LIN {X 0,Y 235.835,Z 423.805,A -85,B 0,C 180,E1 -19803.417,E2 -19803.417} C_VEL
LIN {X 0,Y 235.703,Z 423.051,A -85,B 0,C 180,E1 -19806.85,E2 -19806.85} C_VEL
LIN {X 0,Y 235.515,Z 422.554,A -85,B 0,C 180,E1 -19810.314,E2 -19810.314} C_VEL
LIN {X 0,Y 235.298,Z 422.298,A -85,B 0,C 180,E1 -19815.594,E2 -19815.594} C_VEL
LIN {X 0,Y 235.25,Z 422.493,A -85,B 0,C 180,E1 -19819.185,E2 -19819.185} C_VEL
LIN {X 0,Y 235.278,Z 422.982,A -85,B 0,C 180,E1 -19822.85,E2 -19822.85} C_VEL
LIN {X 0,Y 235.447,Z 423.795,A -85,B 0,C 180,E1 -19826.599,E2 -19826.599} C_VEL
LIN {X 0,Y 235.628,Z 425.005,A -85,B 0,C 180,E1 -19830.468,E2 -19830.468} C_VEL
LIN {X 0,Y 235.886,Z 426.642,A -85,B 0,C 180,E1 -19834.478,E2 -19834.478} C_VEL
LIN {X 0,Y 236.287,Z 428.755,A -85,B 0,C 180,E1 -19838.654,E2 -19838.654} C_VEL
LIN {X 0,Y 236.714,Z 431.464,A -85,B 0,C 180,E1 -19843.068,E2 -19843.068} C_VEL
LIN {X 0,Y 237.092,Z 434.077,A -85,B 0,C 180,E1 -19846.755,E2 -19846.755} C_VEL
LIN {X 0,Y 236.452,Z 434.99,A -85,B 0,C 180,E1 -19847.745,E2 -19847.745} C_VEL
LIN {X 0,Y 233.535,Z 436.791,A -85,B 0,C 180,E1 -19849.288,E2 -19849.288} C_VEL
LIN {X 0,Y 231.568,Z 438.74,A -85,B 0,C 180,E1 -19850.423,E2 -19850.423} C_VEL
LIN {X 0,Y 231.219,Z 440.688,A -85,B 0,C 180,E1 -19851.144,E2 -19851.144} C_VEL
LIN {X 0,Y 231.538,Z 441.777,A -85,B 0,C 180,E1 -19851.419,E2 -19851.419} C_VEL
LIN {X 0,Y 233.164,Z 444.382,A -85,B 0,C 180,E1 -19852.096,E2 -19852.096} C_VEL
LIN {X 0,Y 234.865,Z 448.477,A -85,B 0,C 180,E1 -19852.928,E2 -19852.928} C_VEL
LIN {X 0,Y 238.368,Z 459.348,A -85,B 0,C 180,E1 -19854.983,E2 -19854.983} C_VEL
LIN {X 0,Y 240.952,Z 471.053,A -85,B 0,C 180,E1 -19857.113,E2 -19857.113} C_VEL
LIN {X 0,Y 242.241,Z 482.421,A -85,B 0,C 180,E1 -19859.209,E2 -19859.209} C_VEL
LIN {X 0,Y 242.29,Z 492.215,A -85,B 0,C 180,E1 -19861.082,E2 -19861.082} C_VEL
LIN {X 0,Y 241.351,Z 502.224,A -85,B 0,C 180,E1 -19863.171,E2 -19863.171} C_VEL
LIN {X 0,Y 238.276,Z 511.359,A -85,B 0,C 180,E1 -19865.147,E2 -19865.147} C_VEL
LIN {X 0,Y 234.943,Z 520.47,A -85,B 0,C 180,E1 -19867.627,E2 -19867.627} C_VEL
LIN {X 0,Y 232.548,Z 527.17,A -85,B 0,C 180,E1 -19869.927,E2 -19869.927} C_VEL
LIN {X 0,Y 230.615,Z 532.669,A -85,B 0,C 180,E1 -19872.258,E2 -19872.258} C_VEL
LIN {X 0,Y 228.592,Z 537.603,A -85,B 0,C 180,E1 -19874.852,E2 -19874.852} C_VEL
LIN {X 0,Y 227.248,Z 541.454,A -85,B 0,C 180,E1 -19877.498,E2 -19877.498} C_VEL
LIN {X 0,Y 226.134,Z 545.093,A -85,B 0,C 180,E1 -19881.061,E2 -19881.061} C_VEL
LIN {X 0,Y 225.809,Z 546.282,A -85,B 0,C 180,E1 -19882.849,E2 -19882.849} C_VEL
LIN {X 0,Y 225.616,Z 547.462,A -85,B 0,C 180,E1 -19886.429,E2 -19886.429} C_VEL
LIN {X 0,Y 225.724,Z 547.477,A -85,B 0,C 180,E1 -19888.216,E2 -19888.216} C_VEL
LIN {X 0,Y 225.822,Z 547.081,A -85,B 0,C 180,E1 -19890.001,E2 -19890.001} C_VEL
LIN {X 0,Y 225.761,Z 546.237,A -85,B 0,C 180,E1 -19891.785,E2 -19891.785} C_VEL
LIN {X 0,Y 225.69,Z 543.87,A -85,B 0,C 180,E1 -19894.804,E2 -19894.804} C_VEL
LIN {X 0,Y 225.997,Z 539.926,A -85,B 0,C 180,E1 -19898.045,E2 -19898.045} C_VEL
LIN {X 0,Y 226.529,Z 535.424,A -85,B 0,C 180,E1 -19900.729,E2 -19900.729} C_VEL
LIN {X 0,Y 227.558,Z 528.552,A -85,B 0,C 180,E1 -19903.849,E2 -19903.849} C_VEL
LIN {X 0,Y 228.989,Z 521.094,A -85,B 0,C 180,E1 -19906.493,E2 -19906.493} C_VEL
LIN {X 0,Y 230.359,Z 514.102,A -85,B 0,C 180,E1 -19908.511,E2 -19908.511} C_VEL
LIN {X 0,Y 232.274,Z 504.292,A -85,B 0,C 180,E1 -19910.826,E2 -19910.826} C_VEL
LIN {X 0,Y 234.102,Z 494.094,A -85,B 0,C 180,E1 -19912.739,E2 -19912.739} C_VEL
LIN {X 0,Y 233.818,Z 485.538,A -85,B 0,C 180,E1 -19914.176,E2 -19914.176} C_VEL
LIN {X 0,Y 232.831,Z 472.863,A -85,B 0,C 180,E1 -19915.956,E2 -19915.956} C_VEL
LIN {X 0,Y 231.334,Z 461.288,A -85,B 0,C 180,E1 -19917.299,E2 -19917.299} C_VEL
LIN {X 0,Y 229.017,Z 447.664,A -85,B 0,C 180,E1 -19918.561,E2 -19918.561} C_VEL
LIN {X 0,Y 227.915,Z 441.655,A -85,B 0,C 180,E1 -19919.046,E2 -19919.046} C_VEL
LIN {X 0,Y 229.11,Z 436.101,A -85,B 0,C 180,E1 -19924.082,E2 -19924.082} C_VEL
LIN {X 0,Y 229.433,Z 434.463,A -85,B 0,C 180,E1 -19925.592,E2 -19925.592} C_VEL
LIN {X 0,Y 229.5,Z 431.075,A -85,B 0,C 180,E1 -19928.855,E2 -19928.855} C_VEL
LIN {X 0,Y 228.877,Z 427.486,A -85,B 0,C 180,E1 -19932.527,E2 -19932.527} C_VEL
LIN {X 0,Y 228.1,Z 423.047,A -85,B 0,C 180,E1 -19937.324,E2 -19937.324} C_VEL
LIN {X 0,Y 227.902,Z 422.101,A -85,B 0,C 180,E1 -19938.661,E2 -19938.661} C_VEL
LIN {X 0,Y 227.892,Z 422.093,A -85,B 0,C 180,E1 -19943.304,E2 -19943.304} C_VEL
LIN {X 0,Y 227.881,Z 422.097,A -85,B 0,C 180,E1 -19946.377,E2 -19946.377} C_VEL
LIN {X 0,Y 227.921,Z 422.092,A -85,B 0,C 180,E1 -19950.438,E2 -19950.438} C_VEL
LIN {X 0,Y 227.931,Z 422.086,A -85,B 0,C 180,E1 -19954.426,E2 -19954.426} C_VEL
LIN {X 0,Y 227.964,Z 422.087,A -85,B 0,C 180,E1 -19958.287,E2 -19958.287} C_VEL
LIN {X 0,Y 228.037,Z 422.078,A -85,B 0,C 180,E1 -19962.826,E2 -19962.826} C_VEL
LIN {X 0,Y 228.096,Z 422.068,A -85,B 0,C 180,E1 -19967.544,E2 -19967.544} C_VEL
LIN {X 0,Y 228.309,Z 422.046,A -85,B 0,C 180,E1 -19971.146,E2 -19971.146} C_VEL
LIN {X 0,Y 228.357,Z 422.041,A -85,B 0,C 180,E1 -19972.928,E2 -19972.928} C_VEL
LIN {X 0,Y 228.556,Z 422.01,A -85,B 0,C 180,E1 -19978.238,E2 -19978.238} C_VEL
LIN {X 0,Y 228.556,Z 422.011,A -85,B 0,C 180,E1 -19981.762,E2 -19981.762} C_VEL
LIN {X 0,Y 228.357,Z 422.039,A -85,B 0,C 180,E1 -19987.071,E2 -19987.071} C_VEL
LIN {X 0,Y 228.165,Z 422.063,A -85,B 0,C 180,E1 -19990.65,E2 -19990.65} C_VEL
LIN {X 0,Y 228.066,Z 422.068,A -85,B 0,C 180,E1 -19994.272,E2 -19994.272} C_VEL
LIN {X 0,Y 228.005,Z 422.061,A -85,B 0,C 180,E1 -19997.953,E2 -19997.953} C_VEL
LIN {X 0,Y 227.932,Z 422.085,A -85,B 0,C 180,E1 -20002.329,E2 -20002.329} C_VEL
LIN {X 0,Y 227.945,Z 422.092,A -85,B 0,C 180,E1 -20006.603,E2 -20006.603} C_VEL
LIN {X 0,Y 227.91,Z 422.093,A -85,B 0,C 180,E1 -20010.296,E2 -20010.296} C_VEL
LIN {X 0,Y 227.878,Z 422.087,A -85,B 0,C 180,E1 -20013.72,E2 -20013.72} C_VEL
LIN {X 0,Y 227.845,Z 422.092,A -85,B 0,C 180,E1 -20018.091,E2 -20018.091} C_VEL
LIN {X 0,Y 227.807,Z 422.109,A -85,B 0,C 180,E1 -20022.743,E2 -20022.743} C_VEL
LIN {X 0,Y 227.809,Z 422.103,A -85,B 0,C 180,E1 -20027.257,E2 -20027.257} C_VEL
LIN {X 0,Y 227.872,Z 422.088,A -85,B 0,C 180,E1 -20031.914,E2 -20031.914} C_VEL
LIN {X 0,Y 227.892,Z 422.098,A -85,B 0,C 180,E1 -20036.373,E2 -20036.373} C_VEL
LIN {X 0,Y 227.92,Z 422.092,A -85,B 0,C 180,E1 -20040.437,E2 -20040.437} C_VEL
LIN {X 0,Y 227.931,Z 422.088,A -85,B 0,C 180,E1 -20044.426,E2 -20044.426} C_VEL
LIN {X 0,Y 227.965,Z 422.09,A -85,B 0,C 180,E1 -20048.287,E2 -20048.287} C_VEL
LIN {X 0,Y 228.037,Z 422.079,A -85,B 0,C 180,E1 -20052.825,E2 -20052.825} C_VEL
LIN {X 0,Y 228.096,Z 422.071,A -85,B 0,C 180,E1 -20057.544,E2 -20057.544} C_VEL
LIN {X 0,Y 228.327,Z 422.042,A -85,B 0,C 180,E1 -20061.146,E2 -20061.146} C_VEL
LIN {X 0,Y 228.36,Z 422.037,A -85,B 0,C 180,E1 -20062.928,E2 -20062.928} C_VEL
LIN {X 0,Y 228.556,Z 422.014,A -85,B 0,C 180,E1 -20068.237,E2 -20068.237} C_VEL
LIN {X 0,Y 228.552,Z 422.016,A -85,B 0,C 180,E1 -20071.761,E2 -20071.761} C_VEL
LIN {X 0,Y 228.04,Z 422.078,A -85,B 0,C 180,E1 -20077.081,E2 -20077.081} C_VEL
LIN {X 0,Y 227.754,Z 422.115,A -85,B 0,C 180,E1 -20079.086,E2 -20079.086} C_VEL
LIN {X 0,Y 227.174,Z 425.868,A -85,B 0,C 180,E1 -20083.986,E2 -20083.986} C_VEL
LIN {X 0,Y 231.055,Z 440.646,A -85,B 0,C 180,E1 -20085.434,E2 -20085.434} C_VEL
LIN {X 0,Y 233.596,Z 452.509,A -85,B 0,C 180,E1 -20086.832,E2 -20086.832} C_VEL
LIN {X 0,Y 235.617,Z 464.141,A -85,B 0,C 180,E1 -20088.476,E2 -20088.476} C_VEL
LIN {X 0,Y 236.138,Z 469.588,A -85,B 0,C 180,E1 -20089.335,E2 -20089.335} C_VEL
LIN {X 0,Y 234.409,Z 480.31,A -85,B 0,C 180,E1 -20091.086,E2 -20091.086} C_VEL
LIN {X 0,Y 232.52,Z 490.435,A -85,B 0,C 180,E1 -20093.136,E2 -20093.136} C_VEL
LIN {X 0,Y 230.855,Z 498.791,A -85,B 0,C 180,E1 -20095.226,E2 -20095.226} C_VEL
LIN {X 0,Y 229.203,Z 507.289,A -85,B 0,C 180,E1 -20097.877,E2 -20097.877} C_VEL
LIN {X 0,Y 227.949,Z 513.581,A -85,B 0,C 180,E1 -20100.313,E2 -20100.313} C_VEL
LIN {X 0,Y 226.853,Z 519.558,A -85,B 0,C 180,E1 -20103.231,E2 -20103.231} C_VEL
LIN {X 0,Y 226.113,Z 524.157,A -85,B 0,C 180,E1 -20106.195,E2 -20106.195} C_VEL
LIN {X 0,Y 225.615,Z 527.162,A -85,B 0,C 180,E1 -20108.853,E2 -20108.853} C_VEL
LIN {X 0,Y 225.396,Z 529.228,A -85,B 0,C 180,E1 -20111.553,E2 -20111.553} C_VEL
LIN {X 0,Y 225.352,Z 530.335,A -85,B 0,C 180,E1 -20114.168,E2 -20114.168} C_VEL
LIN {X 0,Y 225.607,Z 530.602,A -85,B 0,C 180,E1 -20116.738,E2 -20116.738} C_VEL
LIN {X 0,Y 226.118,Z 530.085,A -85,B 0,C 180,E1 -20119.254,E2 -20119.254} C_VEL
LIN {X 0,Y 226.867,Z 528.825,A -85,B 0,C 180,E1 -20121.715,E2 -20121.715} C_VEL
LIN {X 0,Y 228.412,Z 525.703,A -85,B 0,C 180,E1 -20125.142,E2 -20125.142} C_VEL
LIN {X 0,Y 230.547,Z 520.882,A -85,B 0,C 180,E1 -20128.598,E2 -20128.598} C_VEL
LIN {X 0,Y 232.641,Z 515.942,A -85,B 0,C 180,E1 -20131.171,E2 -20131.171} C_VEL
LIN {X 0,Y 235.692,Z 508.399,A -85,B 0,C 180,E1 -20134.162,E2 -20134.162} C_VEL
LIN {X 0,Y 238.66,Z 500.676,A -85,B 0,C 180,E1 -20136.547,E2 -20136.547} C_VEL
LIN {X 0,Y 241.823,Z 491.575,A -85,B 0,C 180,E1 -20138.781,E2 -20138.781} C_VEL
LIN {X 0,Y 245.108,Z 480.949,A -85,B 0,C 180,E1 -20140.834,E2 -20140.834} C_VEL
LIN {X 0,Y 245.022,Z 475.384,A -85,B 0,C 180,E1 -20142.041,E2 -20142.041} C_VEL
LIN {X 0,Y 243.7,Z 465.791,A -85,B 0,C 180,E1 -20144.1,E2 -20144.1} C_VEL
LIN {X 0,Y 241.397,Z 456.441,A -85,B 0,C 180,E1 -20146.102,E2 -20146.102} C_VEL
LIN {X 0,Y 237.744,Z 445.879,A -85,B 0,C 180,E1 -20148.397,E2 -20148.397} C_VEL
LIN {X 0,Y 233.783,Z 437.563,A -85,B 0,C 180,E1 -20150.374,E2 -20150.374} C_VEL
LIN {X 0,Y 231.854,Z 433.864,A -85,B 0,C 180,E1 -20151.283,E2 -20151.283} C_VEL
LIN {X 0,Y 229.891,Z 430.981,A -85,B 0,C 180,E1 -20152.148,E2 -20152.148} C_VEL
LIN {X 0,Y 229.311,Z 429.114,A -85,B 0,C 180,E1 -20152.516,E2 -20152.516} C_VEL
LIN {X 0,Y 229.299,Z 426.856,A -85,B 0,C 180,E1 -20158.244,E2 -20158.244} C_VEL
LIN {X 0,Y 229.347,Z 426.269,A -85,B 0,C 180,E1 -20160,E2 -20160} C_VEL
LIN {X 0,Y 228.907,Z 425.375,A -85,B 0,C 180,E1 -20163.521,E2 -20163.521} C_VEL
LIN {X 0,Y 228.783,Z 424.648,A -85,B 0,C 180,E1 -20167.058,E2 -20167.058} C_VEL
LIN {X 0,Y 228.578,Z 424.194,A -85,B 0,C 180,E1 -20170.631,E2 -20170.631} C_VEL
LIN {X 0,Y 228.408,Z 424.01,A -85,B 0,C 180,E1 -20176.077,E2 -20176.077} C_VEL
LIN {X 0,Y 228.344,Z 424.262,A -85,B 0,C 180,E1 -20179.789,E2 -20179.789} C_VEL
LIN {X 0,Y 228.417,Z 424.818,A -85,B 0,C 180,E1 -20183.578,E2 -20183.578} C_VEL
LIN {X 0,Y 228.565,Z 425.728,A -85,B 0,C 180,E1 -20187.466,E2 -20187.466} C_VEL
LIN {X 0,Y 228.774,Z 427.042,A -85,B 0,C 180,E1 -20191.483,E2 -20191.483} C_VEL
LIN {X 0,Y 229.06,Z 428.821,A -85,B 0,C 180,E1 -20195.659,E2 -20195.659} C_VEL
LIN {X 0,Y 229.485,Z 431.109,A -85,B 0,C 180,E1 -20200.039,E2 -20200.039} C_VEL
LIN {X 0,Y 229.946,Z 434.016,A -85,B 0,C 180,E1 -20204.666,E2 -20204.666} C_VEL
LIN {X 0,Y 230.259,Z 436.263,A -85,B 0,C 180,E1 -20207.819,E2 -20207.819} C_VEL
LIN {X 0,Y 230.501,Z 438.815,A -85,B 0,C 180,E1 -20210.885,E2 -20210.885} C_VEL
LIN {X 0,Y 231.538,Z 441.777,A -85,B 0,C 180,E1 -20211.419,E2 -20211.419} C_VEL
LIN {X 0,Y 233.041,Z 446.441,A -85,B 0,C 180,E1 -20212.239,E2 -20212.239} C_VEL
LIN {X 0,Y 233.732,Z 451.625,A -85,B 0,C 180,E1 -20212.942,E2 -20212.942} C_VEL
LIN {X 0,Y 233.917,Z 462.354,A -85,B 0,C 180,E1 -20214.29,E2 -20214.29} C_VEL
LIN {X 0,Y 234.213,Z 467.417,A -85,B 0,C 180,E1 -20215.082,E2 -20215.082} C_VEL
LIN {X 0,Y 234.461,Z 468.99,A -85,B 0,C 180,E1 -20215.38,E2 -20215.38} C_VEL
LIN {X 0,Y 235.858,Z 478.402,A -85,B 0,C 180,E1 -20217.22,E2 -20217.22} C_VEL
LIN {X 0,Y 236.337,Z 487.526,A -85,B 0,C 180,E1 -20219.049,E2 -20219.049} C_VEL
LIN {X 0,Y 235.81,Z 497.788,A -85,B 0,C 180,E1 -20221.194,E2 -20221.194} C_VEL
LIN {X 0,Y 235.062,Z 503.127,A -85,B 0,C 180,E1 -20222.393,E2 -20222.393} C_VEL
LIN {X 0,Y 231.906,Z 512.029,A -85,B 0,C 180,E1 -20224.416,E2 -20224.416} C_VEL
LIN {X 0,Y 228.479,Z 520.817,A -85,B 0,C 180,E1 -20226.91,E2 -20226.91} C_VEL
LIN {X 0,Y 225.831,Z 527.661,A -85,B 0,C 180,E1 -20229.377,E2 -20229.377} C_VEL
LIN {X 0,Y 223.854,Z 532.868,A -85,B 0,C 180,E1 -20231.703,E2 -20231.703} C_VEL
LIN {X 0,Y 221.737,Z 537.702,A -85,B 0,C 180,E1 -20234.372,E2 -20234.372} C_VEL
LIN {X 0,Y 220.275,Z 541.458,A -85,B 0,C 180,E1 -20237.096,E2 -20237.096} C_VEL
LIN {X 0,Y 219.602,Z 543.43,A -85,B 0,C 180,E1 -20238.93,E2 -20238.93} C_VEL
LIN {X 0,Y 219.087,Z 544.981,A -85,B 0,C 180,E1 -20240.771,E2 -20240.771} C_VEL
LIN {X 0,Y 218.568,Z 546.843,A -85,B 0,C 180,E1 -20244.465,E2 -20244.465} C_VEL
LIN {X 0,Y 218.635,Z 547.175,A -85,B 0,C 180,E1 -20248.159,E2 -20248.159} C_VEL
LIN {X 0,Y 218.754,Z 546.708,A -85,B 0,C 180,E1 -20250.001,E2 -20250.001} C_VEL
LIN {X 0,Y 218.671,Z 545.825,A -85,B 0,C 180,E1 -20251.842,E2 -20251.842} C_VEL
LIN {X 0,Y 218.593,Z 543.659,A -85,B 0,C 180,E1 -20254.664,E2 -20254.664} C_VEL
LIN {X 0,Y 218.813,Z 540.59,A -85,B 0,C 180,E1 -20257.382,E2 -20257.382} C_VEL
LIN {X 0,Y 219.292,Z 536.374,A -85,B 0,C 180,E1 -20260.153,E2 -20260.153} C_VEL
LIN {X 0,Y 220.229,Z 529.927,A -85,B 0,C 180,E1 -20263.378,E2 -20263.378} C_VEL
LIN {X 0,Y 221.655,Z 522.877,A -85,B 0,C 180,E1 -20266.108,E2 -20266.108} C_VEL
LIN {X 0,Y 223.291,Z 514.581,A -85,B 0,C 180,E1 -20268.665,E2 -20268.665} C_VEL
LIN {X 0,Y 225.195,Z 505.019,A -85,B 0,C 180,E1 -20271.033,E2 -20271.033} C_VEL
LIN {X 0,Y 227.088,Z 495.116,A -85,B 0,C 180,E1 -20273,E2 -20273} C_VEL
LIN {X 0,Y 227.041,Z 488.306,A -85,B 0,C 180,E1 -20274.207,E2 -20274.207} C_VEL
LIN {X 0,Y 226.276,Z 476.943,A -85,B 0,C 180,E1 -20275.972,E2 -20275.972} C_VEL
LIN {X 0,Y 224.921,Z 464.647,A -85,B 0,C 180,E1 -20277.548,E2 -20277.548} C_VEL
LIN {X 0,Y 222.726,Z 450.893,A -85,B 0,C 180,E1 -20278.964,E2 -20278.964} C_VEL
LIN {X 0,Y 221.002,Z 441.394,A -85,B 0,C 180,E1 -20279.779,E2 -20279.779} C_VEL
LIN {X 0,Y 222.16,Z 436.145,A -85,B 0,C 180,E1 -20284.711,E2 -20284.711} C_VEL
LIN {X 0,Y 222.469,Z 432.936,A -85,B 0,C 180,E1 -20287.835,E2 -20287.835} C_VEL
LIN {X 0,Y 222.174,Z 430.256,A -85,B 0,C 180,E1 -20290.607,E2 -20290.607} C_VEL
LIN {X 0,Y 221.536,Z 426.856,A -85,B 0,C 180,E1 -20294.261,E2 -20294.261} C_VEL
LIN {X 0,Y 220.878,Z 422.977,A -85,B 0,C 180,E1 -20298.787,E2 -20298.787} C_VEL
LIN {X 0,Y 220.826,Z 422.977,A -85,B 0,C 180,E1 -20302.793,E2 -20302.793} C_VEL
LIN {X 0,Y 220.82,Z 422.982,A -85,B 0,C 180,E1 -20307.244,E2 -20307.244} C_VEL
LIN {X 0,Y 220.839,Z 422.97,A -85,B 0,C 180,E1 -20311.487,E2 -20311.487} C_VEL
LIN {X 0,Y 220.87,Z 422.971,A -85,B 0,C 180,E1 -20315.565,E2 -20315.565} C_VEL
LIN {X 0,Y 220.895,Z 422.968,A -85,B 0,C 180,E1 -20319.514,E2 -20319.514} C_VEL
LIN {X 0,Y 221.019,Z 422.954,A -85,B 0,C 180,E1 -20323.37,E2 -20323.37} C_VEL
LIN {X 0,Y 221.114,Z 422.939,A -85,B 0,C 180,E1 -20329.006,E2 -20329.006} C_VEL
LIN {X 0,Y 221.292,Z 422.919,A -85,B 0,C 180,E1 -20332.702,E2 -20332.702} C_VEL
LIN {X 0,Y 221.514,Z 422.887,A -85,B 0,C 180,E1 -20338.182,E2 -20338.182} C_VEL
LIN {X 0,Y 221.514,Z 422.888,A -85,B 0,C 180,E1 -20341.818,E2 -20341.818} C_VEL
LIN {X 0,Y 221.292,Z 422.918,A -85,B 0,C 180,E1 -20347.298,E2 -20347.298} C_VEL
LIN {X 0,Y 221.114,Z 422.94,A -85,B 0,C 180,E1 -20350.994,E2 -20350.994} C_VEL
LIN {X 0,Y 221.018,Z 422.936,A -85,B 0,C 180,E1 -20356.63,E2 -20356.63} C_VEL
LIN {X 0,Y 220.894,Z 422.955,A -85,B 0,C 180,E1 -20360.486,E2 -20360.486} C_VEL
LIN {X 0,Y 220.869,Z 422.969,A -85,B 0,C 180,E1 -20364.435,E2 -20364.435} C_VEL
LIN {X 0,Y 220.839,Z 422.977,A -85,B 0,C 180,E1 -20368.513,E2 -20368.513} C_VEL
LIN {X 0,Y 220.819,Z 422.969,A -85,B 0,C 180,E1 -20372.756,E2 -20372.756} C_VEL
LIN {X 0,Y 220.811,Z 422.967,A -85,B 0,C 180,E1 -20377.278,E2 -20377.278} C_VEL
LIN {X 0,Y 220.796,Z 422.975,A -85,B 0,C 180,E1 -20380.188,E2 -20380.188} C_VEL
LIN {X 0,Y 220.769,Z 422.986,A -85,B 0,C 180,E1 -20384.455,E2 -20384.455} C_VEL
LIN {X 0,Y 220.773,Z 422.979,A -85,B 0,C 180,E1 -20388.048,E2 -20388.048} C_VEL
LIN {X 0,Y 220.834,Z 422.969,A -85,B 0,C 180,E1 -20392.794,E2 -20392.794} C_VEL
LIN {X 0,Y 220.826,Z 422.976,A -85,B 0,C 180,E1 -20397.245,E2 -20397.245} C_VEL
LIN {X 0,Y 220.838,Z 422.969,A -85,B 0,C 180,E1 -20401.486,E2 -20401.486} C_VEL
LIN {X 0,Y 220.87,Z 422.969,A -85,B 0,C 180,E1 -20405.565,E2 -20405.565} C_VEL
LIN {X 0,Y 220.895,Z 422.967,A -85,B 0,C 180,E1 -20409.514,E2 -20409.514} C_VEL
LIN {X 0,Y 221.019,Z 422.951,A -85,B 0,C 180,E1 -20413.37,E2 -20413.37} C_VEL
LIN {X 0,Y 221.119,Z 422.938,A -85,B 0,C 180,E1 -20419.006,E2 -20419.006} C_VEL
LIN {X 0,Y 221.313,Z 422.916,A -85,B 0,C 180,E1 -20422.702,E2 -20422.702} C_VEL
LIN {X 0,Y 221.514,Z 422.89,A -85,B 0,C 180,E1 -20428.181,E2 -20428.181} C_VEL
LIN {X 0,Y 221.508,Z 422.894,A -85,B 0,C 180,E1 -20431.817,E2 -20431.817} C_VEL
LIN {X 0,Y 220.963,Z 422.96,A -85,B 0,C 180,E1 -20437.309,E2 -20437.309} C_VEL
LIN {X 0,Y 220.683,Z 423.074,A -85,B 0,C 180,E1 -20439.162,E2 -20439.162} C_VEL
LIN {X 0,Y 220.175,Z 426.153,A -85,B 0,C 180,E1 -20443.262,E2 -20443.262} C_VEL
LIN {X 0,Y 223.641,Z 439.187,A -85,B 0,C 180,E1 -20444.56,E2 -20444.56} C_VEL
LIN {X 0,Y 226.316,Z 451.122,A -85,B 0,C 180,E1 -20445.997,E2 -20445.997} C_VEL
LIN {X 0,Y 228.418,Z 462.946,A -85,B 0,C 180,E1 -20447.687,E2 -20447.687} C_VEL
LIN {X 0,Y 229.33,Z 469.548,A -85,B 0,C 180,E1 -20448.77,E2 -20448.77} C_VEL
LIN {X 0,Y 227.654,Z 480.216,A -85,B 0,C 180,E1 -20450.557,E2 -20450.557} C_VEL
LIN {X 0,Y 225.684,Z 490.407,A -85,B 0,C 180,E1 -20452.666,E2 -20452.666} C_VEL
LIN {X 0,Y 223.941,Z 498.898,A -85,B 0,C 180,E1 -20454.838,E2 -20454.838} C_VEL
LIN {X 0,Y 222.181,Z 507.691,A -85,B 0,C 180,E1 -20457.663,E2 -20457.663} C_VEL
LIN {X 0,Y 220.66,Z 515.118,A -85,B 0,C 180,E1 -20460.689,E2 -20460.689} C_VEL
LIN {X 0,Y 219.62,Z 520.768,A -85,B 0,C 180,E1 -20463.693,E2 -20463.693} C_VEL
LIN {X 0,Y 218.913,Z 524.943,A -85,B 0,C 180,E1 -20466.621,E2 -20466.621} C_VEL
LIN {X 0,Y 218.374,Z 528.377,A -85,B 0,C 180,E1 -20470.064,E2 -20470.064} C_VEL
LIN {X 0,Y 218.251,Z 529.922,A -85,B 0,C 180,E1 -20472.548,E2 -20472.548} C_VEL
LIN {X 0,Y 218.314,Z 530.772,A -85,B 0,C 180,E1 -20475.089,E2 -20475.089} C_VEL
LIN {X 0,Y 218.659,Z 530.86,A -85,B 0,C 180,E1 -20477.666,E2 -20477.666} C_VEL
LIN {X 0,Y 219.313,Z 530.146,A -85,B 0,C 180,E1 -20480.271,E2 -20480.271} C_VEL
LIN {X 0,Y 220.258,Z 528.623,A -85,B 0,C 180,E1 -20482.909,E2 -20482.909} C_VEL
LIN {X 0,Y 221.527,Z 526.216,A -85,B 0,C 180,E1 -20485.572,E2 -20485.572} C_VEL
LIN {X 0,Y 223.753,Z 521.546,A -85,B 0,C 180,E1 -20489.085,E2 -20489.085} C_VEL
LIN {X 0,Y 226.456,Z 515.596,A -85,B 0,C 180,E1 -20492.256,E2 -20492.256} C_VEL
LIN {X 0,Y 229.341,Z 508.93,A -85,B 0,C 180,E1 -20494.958,E2 -20494.958} C_VEL
LIN {X 0,Y 232.287,Z 501.744,A -85,B 0,C 180,E1 -20497.259,E2 -20497.259} C_VEL
LIN {X 0,Y 235.51,Z 493.129,A -85,B 0,C 180,E1 -20499.474,E2 -20499.474} C_VEL
LIN {X 0,Y 238.667,Z 483.566,A -85,B 0,C 180,E1 -20501.434,E2 -20501.434} C_VEL
LIN {X 0,Y 239.088,Z 481.667,A -85,B 0,C 180,E1 -20501.801,E2 -20501.801} C_VEL
LIN {X 0,Y 238.557,Z 473.342,A -85,B 0,C 180,E1 -20503.747,E2 -20503.747} C_VEL
LIN {X 0,Y 237.059,Z 464.122,A -85,B 0,C 180,E1 -20505.843,E2 -20505.843} C_VEL
LIN {X 0,Y 234.087,Z 453.725,A -85,B 0,C 180,E1 -20508.268,E2 -20508.268} C_VEL
LIN {X 0,Y 231.492,Z 446.805,A -85,B 0,C 180,E1 -20509.947,E2 -20509.947} C_VEL
LIN {X 0,Y 227.917,Z 439.271,A -85,B 0,C 180,E1 -20511.929,E2 -20511.929} C_VEL
LIN {X 0,Y 225.984,Z 436.076,A -85,B 0,C 180,E1 -20512.91,E2 -20512.91} C_VEL
LIN {X 0,Y 225.03,Z 434.44,A -85,B 0,C 180,E1 -20513.387,E2 -20513.387} C_VEL
LIN {X 0,Y 222.916,Z 431.575,A -85,B 0,C 180,E1 -20514.403,E2 -20514.403} C_VEL
LIN {X 0,Y 222.29,Z 429.592,A -85,B 0,C 180,E1 -20514.899,E2 -20514.899} C_VEL
LIN {X 0,Y 222.364,Z 428.394,A -85,B 0,C 180,E1 -20518.189,E2 -20518.189} C_VEL
LIN {X 0,Y 222.415,Z 427.824,A -85,B 0,C 180,E1 -20520,E2 -20520} C_VEL
LIN {X 0,Y 221.969,Z 426.951,A -85,B 0,C 180,E1 -20523.631,E2 -20523.631} C_VEL
LIN {X 0,Y 221.856,Z 426.256,A -85,B 0,C 180,E1 -20527.28,E2 -20527.28} C_VEL
LIN {X 0,Y 221.645,Z 425.849,A -85,B 0,C 180,E1 -20530.968,E2 -20530.968} C_VEL
LIN {X 0,Y 221.503,Z 425.734,A -85,B 0,C 180,E1 -20536.592,E2 -20536.592} C_VEL
LIN {X 0,Y 221.45,Z 426.047,A -85,B 0,C 180,E1 -20540.432,E2 -20540.432} C_VEL
LIN {X 0,Y 221.528,Z 426.682,A -85,B 0,C 180,E1 -20544.358,E2 -20544.358} C_VEL
LIN {X 0,Y 221.695,Z 427.69,A -85,B 0,C 180,E1 -20548.393,E2 -20548.393} C_VEL
LIN {X 0,Y 221.917,Z 429.133,A -85,B 0,C 180,E1 -20552.574,E2 -20552.574} C_VEL
LIN {X 0,Y 222.358,Z 431.469,A -85,B 0,C 180,E1 -20557.8,E2 -20557.8} C_VEL
LIN {X 0,Y 222.669,Z 433.515,A -85,B 0,C 180,E1 -20561.515,E2 -20561.515} C_VEL
LIN {X 0,Y 223.123,Z 436.466,A -85,B 0,C 180,E1 -20566.136,E2 -20566.136} C_VEL
LIN {X 0,Y 223.334,Z 438.161,A -85,B 0,C 180,E1 -20568.52,E2 -20568.52} C_VEL
LIN {X 0,Y 224.515,Z 441.421,A -85,B 0,C 180,E1 -20569.213,E2 -20569.213} C_VEL
LIN {X 0,Y 226.615,Z 444.574,A -85,B 0,C 180,E1 -20570.187,E2 -20570.187} C_VEL
LIN {X 0,Y 228.466,Z 448.596,A -85,B 0,C 180,E1 -20571.171,E2 -20571.171} C_VEL
LIN {X 0,Y 230.722,Z 454.495,A -85,B 0,C 180,E1 -20572.468,E2 -20572.468} C_VEL
LIN {X 0,Y 233.238,Z 463.05,A -85,B 0,C 180,E1 -20574.214,E2 -20574.214} C_VEL
LIN {X 0,Y 234.461,Z 468.99,A -85,B 0,C 180,E1 -20575.38,E2 -20575.38} C_VEL
LIN {X 0,Y 234.759,Z 473.886,A -85,B 0,C 180,E1 -20576.215,E2 -20576.215} C_VEL
LIN {X 0,Y 233.953,Z 479.09,A -85,B 0,C 180,E1 -20576.937,E2 -20576.937} C_VEL
LIN {X 0,Y 231.165,Z 489.229,A -85,B 0,C 180,E1 -20578.37,E2 -20578.37} C_VEL
LIN {X 0,Y 230.115,Z 493.949,A -85,B 0,C 180,E1 -20579.229,E2 -20579.229} C_VEL
LIN {X 0,Y 229.937,Z 495.417,A -85,B 0,C 180,E1 -20579.55,E2 -20579.55} C_VEL
LIN {X 0,Y 228.798,Z 504.005,A -85,B 0,C 180,E1 -20581.569,E2 -20581.569} C_VEL
LIN {X 0,Y 225.553,Z 512.702,A -85,B 0,C 180,E1 -20583.641,E2 -20583.641} C_VEL
LIN {X 0,Y 221.978,Z 521.337,A -85,B 0,C 180,E1 -20586.193,E2 -20586.193} C_VEL
LIN {X 0,Y 219.137,Z 528.2,A -85,B 0,C 180,E1 -20588.795,E2 -20588.795} C_VEL
LIN {X 0,Y 217.12,Z 533.108,A -85,B 0,C 180,E1 -20591.115,E2 -20591.115} C_VEL
LIN {X 0,Y 214.902,Z 537.812,A -85,B 0,C 180,E1 -20593.861,E2 -20593.861} C_VEL
LIN {X 0,Y 213.315,Z 541.464,A -85,B 0,C 180,E1 -20596.667,E2 -20596.667} C_VEL
LIN {X 0,Y 212.609,Z 543.384,A -85,B 0,C 180,E1 -20598.561,E2 -20598.561} C_VEL
LIN {X 0,Y 211.669,Z 545.931,A -85,B 0,C 180,E1 -20602.369,E2 -20602.369} C_VEL
LIN {X 0,Y 211.437,Z 546.946,A -85,B 0,C 180,E1 -20606.189,E2 -20606.189} C_VEL
LIN {X 0,Y 211.547,Z 546.843,A -85,B 0,C 180,E1 -20608.097,E2 -20608.097} C_VEL
LIN {X 0,Y 211.687,Z 546.332,A -85,B 0,C 180,E1 -20610.001,E2 -20610.001} C_VEL
LIN {X 0,Y 211.584,Z 545.41,A -85,B 0,C 180,E1 -20611.904,E2 -20611.904} C_VEL
LIN {X 0,Y 211.508,Z 543.417,A -85,B 0,C 180,E1 -20614.55,E2 -20614.55} C_VEL
LIN {X 0,Y 211.743,Z 540.009,A -85,B 0,C 180,E1 -20617.63,E2 -20617.63} C_VEL
LIN {X 0,Y 212.269,Z 535.701,A -85,B 0,C 180,E1 -20620.493,E2 -20620.493} C_VEL
LIN {X 0,Y 213.078,Z 530.167,A -85,B 0,C 180,E1 -20623.35,E2 -20623.35} C_VEL
LIN {X 0,Y 214.527,Z 523.266,A -85,B 0,C 180,E1 -20626.169,E2 -20626.169} C_VEL
LIN {X 0,Y 216.293,Z 514.598,A -85,B 0,C 180,E1 -20628.962,E2 -20628.962} C_VEL
LIN {X 0,Y 218.113,Z 505.73,A -85,B 0,C 180,E1 -20631.254,E2 -20631.254} C_VEL
LIN {X 0,Y 220.25,Z 494.853,A -85,B 0,C 180,E1 -20633.508,E2 -20633.508} C_VEL
LIN {X 0,Y 219.875,Z 484.523,A -85,B 0,C 180,E1 -20635.372,E2 -20635.372} C_VEL
LIN {X 0,Y 219.032,Z 473.317,A -85,B 0,C 180,E1 -20637.07,E2 -20637.07} C_VEL
LIN {X 0,Y 217.436,Z 460.354,A -85,B 0,C 180,E1 -20638.69,E2 -20638.69} C_VEL
LIN {X 0,Y 215.113,Z 447.007,A -85,B 0,C 180,E1 -20640.016,E2 -20640.016} C_VEL
LIN {X 0,Y 214.084,Z 441.156,A -85,B 0,C 180,E1 -20640.516,E2 -20640.516} C_VEL
LIN {X 0,Y 215.194,Z 436.293,A -85,B 0,C 180,E1 -20645.267,E2 -20645.267} C_VEL
LIN {X 0,Y 215.402,Z 433.154,A -85,B 0,C 180,E1 -20648.458,E2 -20648.458} C_VEL
LIN {X 0,Y 215.022,Z 430.532,A -85,B 0,C 180,E1 -20651.257,E2 -20651.257} C_VEL
LIN {X 0,Y 214.361,Z 427.072,A -85,B 0,C 180,E1 -20655.146,E2 -20655.146} C_VEL
LIN {X 0,Y 213.799,Z 423.86,A -85,B 0,C 180,E1 -20659.118,E2 -20659.118} C_VEL
LIN {X 0,Y 213.746,Z 423.852,A -85,B 0,C 180,E1 -20663.712,E2 -20663.712} C_VEL
LIN {X 0,Y 213.797,Z 423.855,A -85,B 0,C 180,E1 -20668.725,E2 -20668.725} C_VEL
LIN {X 0,Y 213.828,Z 423.841,A -85,B 0,C 180,E1 -20672.603,E2 -20672.603} C_VEL
LIN {X 0,Y 213.854,Z 423.846,A -85,B 0,C 180,E1 -20676.953,E2 -20676.953} C_VEL
LIN {X 0,Y 213.946,Z 423.832,A -85,B 0,C 180,E1 -20682.804,E2 -20682.804} C_VEL
LIN {X 0,Y 213.983,Z 423.83,A -85,B 0,C 180,E1 -20686.708,E2 -20686.708} C_VEL
LIN {X 0,Y 214.17,Z 423.804,A -85,B 0,C 180,E1 -20690.556,E2 -20690.556} C_VEL
LIN {X 0,Y 214.23,Z 423.798,A -85,B 0,C 180,E1 -20692.46,E2 -20692.46} C_VEL
LIN {X 0,Y 214.447,Z 423.767,A -85,B 0,C 180,E1 -20698.122,E2 -20698.122} C_VEL
LIN {X 0,Y 214.548,Z 423.757,A -85,B 0,C 180,E1 -20700,E2 -20700} C_VEL
LIN {X 0,Y 214.447,Z 423.769,A -85,B 0,C 180,E1 -20701.878,E2 -20701.878} C_VEL
LIN {X 0,Y 214.23,Z 423.796,A -85,B 0,C 180,E1 -20707.54,E2 -20707.54} C_VEL
LIN {X 0,Y 214.047,Z 423.818,A -85,B 0,C 180,E1 -20711.362,E2 -20711.362} C_VEL
LIN {X 0,Y 213.935,Z 423.822,A -85,B 0,C 180,E1 -20715.237,E2 -20715.237} C_VEL
LIN {X 0,Y 213.842,Z 423.829,A -85,B 0,C 180,E1 -20719.187,E2 -20719.187} C_VEL
LIN {X 0,Y 213.849,Z 423.843,A -85,B 0,C 180,E1 -20723.227,E2 -20723.227} C_VEL
LIN {X 0,Y 213.831,Z 423.848,A -85,B 0,C 180,E1 -20727.45,E2 -20727.45} C_VEL
LIN {X 0,Y 213.779,Z 423.848,A -85,B 0,C 180,E1 -20731.736,E2 -20731.736} C_VEL
LIN {X 0,Y 213.745,Z 423.838,A -85,B 0,C 180,E1 -20736.288,E2 -20736.288} C_VEL
LIN {X 0,Y 213.712,Z 423.861,A -85,B 0,C 180,E1 -20741.125,E2 -20741.125} C_VEL
LIN {X 0,Y 213.704,Z 423.863,A -85,B 0,C 180,E1 -20743.679,E2 -20743.679} C_VEL
LIN {X 0,Y 213.704,Z 423.864,A -85,B 0,C 180,E1 -20746.345,E2 -20746.345} C_VEL
LIN {X 0,Y 213.737,Z 423.847,A -85,B 0,C 180,E1 -20751.336,E2 -20751.336} C_VEL
LIN {X 0,Y 213.771,Z 423.854,A -85,B 0,C 180,E1 -20756.02,E2 -20756.02} C_VEL
LIN {X 0,Y 213.782,Z 423.853,A -85,B 0,C 180,E1 -20760.454,E2 -20760.454} C_VEL
LIN {X 0,Y 213.804,Z 423.849,A -85,B 0,C 180,E1 -20764.701,E2 -20764.701} C_VEL
LIN {X 0,Y 213.816,Z 423.85,A -85,B 0,C 180,E1 -20768.803,E2 -20768.803} C_VEL
LIN {X 0,Y 213.946,Z 423.834,A -85,B 0,C 180,E1 -20772.803,E2 -20772.803} C_VEL
LIN {X 0,Y 213.983,Z 423.831,A -85,B 0,C 180,E1 -20776.708,E2 -20776.708} C_VEL
LIN {X 0,Y 214.199,Z 423.805,A -85,B 0,C 180,E1 -20780.557,E2 -20780.557} C_VEL
LIN {X 0,Y 214.25,Z 423.797,A -85,B 0,C 180,E1 -20782.46,E2 -20782.46} C_VEL
LIN {X 0,Y 214.447,Z 423.77,A -85,B 0,C 180,E1 -20788.121,E2 -20788.121} C_VEL
LIN {X 0,Y 214.551,Z 423.762,A -85,B 0,C 180,E1 -20789.999,E2 -20789.999} C_VEL
LIN {X 0,Y 214.44,Z 423.774,A -85,B 0,C 180,E1 -20791.877,E2 -20791.877} C_VEL
LIN {X 0,Y 213.894,Z 423.84,A -85,B 0,C 180,E1 -20797.551,E2 -20797.551} C_VEL
LIN {X 0,Y 213.627,Z 424.046,A -85,B 0,C 180,E1 -20799.265,E2 -20799.265} C_VEL
LIN {X 0,Y 213.177,Z 426.423,A -85,B 0,C 180,E1 -20802.494,E2 -20802.494} C_VEL
LIN {X 0,Y 217.086,Z 441.141,A -85,B 0,C 180,E1 -20804.052,E2 -20804.052} C_VEL
LIN {X 0,Y 219.678,Z 452.86,A -85,B 0,C 180,E1 -20805.541,E2 -20805.541} C_VEL
LIN {X 0,Y 221.665,Z 464.481,A -85,B 0,C 180,E1 -20807.291,E2 -20807.291} C_VEL
LIN {X 0,Y 222.437,Z 471.003,A -85,B 0,C 180,E1 -20808.418,E2 -20808.418} C_VEL
LIN {X 0,Y 220.623,Z 481.552,A -85,B 0,C 180,E1 -20810.268,E2 -20810.268} C_VEL
LIN {X 0,Y 218.653,Z 491.445,A -85,B 0,C 180,E1 -20812.416,E2 -20812.416} C_VEL
LIN {X 0,Y 216.692,Z 500.689,A -85,B 0,C 180,E1 -20814.937,E2 -20814.937} C_VEL
LIN {X 0,Y 215.068,Z 508.475,A -85,B 0,C 180,E1 -20817.577,E2 -20817.577} C_VEL
LIN {X 0,Y 213.697,Z 514.916,A -85,B 0,C 180,E1 -20820.293,E2 -20820.293} C_VEL
LIN {X 0,Y 212.695,Z 520.051,A -85,B 0,C 180,E1 -20823.01,E2 -20823.01} C_VEL
LIN {X 0,Y 211.795,Z 525.251,A -85,B 0,C 180,E1 -20826.675,E2 -20826.675} C_VEL
LIN {X 0,Y 211.285,Z 528.555,A -85,B 0,C 180,E1 -20830.088,E2 -20830.088} C_VEL
LIN {X 0,Y 211.14,Z 530.265,A -85,B 0,C 180,E1 -20832.921,E2 -20832.921} C_VEL
LIN {X 0,Y 211.285,Z 531.09,A -85,B 0,C 180,E1 -20835.691,E2 -20835.691} C_VEL
LIN {X 0,Y 212.031,Z 530.836,A -85,B 0,C 180,E1 -20839.671,E2 -20839.671} C_VEL
LIN {X 0,Y 212.932,Z 529.638,A -85,B 0,C 180,E1 -20842.384,E2 -20842.384} C_VEL
LIN {X 0,Y 214.743,Z 526.557,A -85,B 0,C 180,E1 -20846.195,E2 -20846.195} C_VEL
LIN {X 0,Y 217.087,Z 522.051,A -85,B 0,C 180,E1 -20849.727,E2 -20849.727} C_VEL
LIN {X 0,Y 219.843,Z 516.42,A -85,B 0,C 180,E1 -20852.885,E2 -20852.885} C_VEL
LIN {X 0,Y 223.221,Z 509.122,A -85,B 0,C 180,E1 -20855.928,E2 -20855.928} C_VEL
LIN {X 0,Y 226.638,Z 501.223,A -85,B 0,C 180,E1 -20858.478,E2 -20858.478} C_VEL
LIN {X 0,Y 230.434,Z 491.296,A -85,B 0,C 180,E1 -20860.988,E2 -20860.988} C_VEL
LIN {X 0,Y 232.865,Z 484.289,A -85,B 0,C 180,E1 -20862.434,E2 -20862.434} C_VEL
LIN {X 0,Y 232.744,Z 476.985,A -85,B 0,C 180,E1 -20864.231,E2 -20864.231} C_VEL
LIN {X 0,Y 231.604,Z 468.053,A -85,B 0,C 180,E1 -20866.398,E2 -20866.398} C_VEL
LIN {X 0,Y 229.109,Z 458.055,A -85,B 0,C 180,E1 -20868.907,E2 -20868.907} C_VEL
LIN {X 0,Y 225.674,Z 448.377,A -85,B 0,C 180,E1 -20871.445,E2 -20871.445} C_VEL
LIN {X 0,Y 221.431,Z 440.186,A -85,B 0,C 180,E1 -20873.965,E2 -20873.965} C_VEL
LIN {X 0,Y 219.249,Z 436.795,A -85,B 0,C 180,E1 -20875.211,E2 -20875.211} C_VEL
LIN {X 0,Y 218.487,Z 435.333,A -85,B 0,C 180,E1 -20875.671,E2 -20875.671} C_VEL
LIN {X 0,Y 216.276,Z 432.694,A -85,B 0,C 180,E1 -20876.857,E2 -20876.857} C_VEL
LIN {X 0,Y 215.382,Z 430.14,A -85,B 0,C 180,E1 -20877.546,E2 -20877.546} C_VEL
LIN {X 0,Y 215.508,Z 429.371,A -85,B 0,C 180,E1 -20880,E2 -20880} C_VEL
LIN {X 0,Y 215.037,Z 428.538,A -85,B 0,C 180,E1 -20883.748,E2 -20883.748} C_VEL
LIN {X 0,Y 214.926,Z 427.872,A -85,B 0,C 180,E1 -20887.516,E2 -20887.516} C_VEL
LIN {X 0,Y 214.715,Z 427.506,A -85,B 0,C 180,E1 -20891.326,E2 -20891.326} C_VEL
LIN {X 0,Y 214.583,Z 427.422,A -85,B 0,C 180,E1 -20895.19,E2 -20895.19} C_VEL
LIN {X 0,Y 214.548,Z 427.634,A -85,B 0,C 180,E1 -20899.122,E2 -20899.122} C_VEL
LIN {X 0,Y 214.637,Z 428.242,A -85,B 0,C 180,E1 -20903.537,E2 -20903.537} C_VEL
LIN {X 0,Y 214.782,Z 429.258,A -85,B 0,C 180,E1 -20907.937,E2 -20907.937} C_VEL
LIN {X 0,Y 214.969,Z 430.494,A -85,B 0,C 180,E1 -20911.788,E2 -20911.788} C_VEL
LIN {X 0,Y 215.234,Z 432.211,A -85,B 0,C 180,E1 -20915.998,E2 -20915.998} C_VEL
LIN {X 0,Y 215.686,Z 434.544,A -85,B 0,C 180,E1 -20920.669,E2 -20920.669} C_VEL
LIN {X 0,Y 216.116,Z 437.631,A -85,B 0,C 180,E1 -20925.748,E2 -20925.748} C_VEL
LIN {X 0,Y 217.425,Z 441.015,A -85,B 0,C 180,E1 -20926.629,E2 -20926.629} C_VEL
LIN {X 0,Y 219.699,Z 444.17,A -85,B 0,C 180,E1 -20927.83,E2 -20927.83} C_VEL
LIN {X 0,Y 221.426,Z 447.891,A -85,B 0,C 180,E1 -20928.861,E2 -20928.861} C_VEL
LIN {X 0,Y 222.698,Z 450.113,A -85,B 0,C 180,E1 -20929.54,E2 -20929.54} C_VEL
LIN {X 0,Y 225.744,Z 457.855,A -85,B 0,C 180,E1 -20931.491,E2 -20931.491} C_VEL
LIN {X 0,Y 228.199,Z 467.369,A -85,B 0,C 180,E1 -20933.571,E2 -20933.571} C_VEL
LIN {X 0,Y 229.877,Z 478.673,A -85,B 0,C 180,E1 -20935.957,E2 -20935.957} C_VEL
LIN {X 0,Y 230.32,Z 488.518,A -85,B 0,C 180,E1 -20938.037,E2 -20938.037} C_VEL
LIN {X 0,Y 229.937,Z 495.417,A -85,B 0,C 180,E1 -20939.55,E2 -20939.55} C_VEL
LIN {X 0,Y 229.312,Z 498.428,A -85,B 0,C 180,E1 -20940.171,E2 -20940.171} C_VEL
LIN {X 0,Y 228.066,Z 501.453,A -85,B 0,C 180,E1 -20940.727,E2 -20940.727} C_VEL
LIN {X 0,Y 224.459,Z 507.306,A -85,B 0,C 180,E1 -20941.741,E2 -20941.741} C_VEL
LIN {X 0,Y 219.444,Z 514.276,A -85,B 0,C 180,E1 -20943.126,E2 -20943.126} C_VEL
LIN {X 0,Y 217.207,Z 518.115,A -85,B 0,C 180,E1 -20944.195,E2 -20944.195} C_VEL
LIN {X 0,Y 213.538,Z 526.294,A -85,B 0,C 180,E1 -20947.153,E2 -20947.153} C_VEL
LIN {X 0,Y 210.412,Z 533.356,A -85,B 0,C 180,E1 -20950.488,E2 -20950.488} C_VEL
LIN {X 0,Y 208.089,Z 537.951,A -85,B 0,C 180,E1 -20953.318,E2 -20953.318} C_VEL
LIN {X 0,Y 206.372,Z 541.496,A -85,B 0,C 180,E1 -20956.21,E2 -20956.21} C_VEL
LIN {X 0,Y 205.052,Z 544.728,A -85,B 0,C 180,E1 -20960.133,E2 -20960.133} C_VEL
LIN {X 0,Y 204.4,Z 546.416,A -85,B 0,C 180,E1 -20964.08,E2 -20964.08} C_VEL
LIN {X 0,Y 204.337,Z 546.664,A -85,B 0,C 180,E1 -20966.056,E2 -20966.056} C_VEL
LIN {X 0,Y 204.461,Z 546.5,A -85,B 0,C 180,E1 -20968.031,E2 -20968.031} C_VEL
LIN {X 0,Y 204.621,Z 545.947,A -85,B 0,C 180,E1 -20970.001,E2 -20970.001} C_VEL
LIN {X 0,Y 204.498,Z 544.979,A -85,B 0,C 180,E1 -20971.97,E2 -20971.97} C_VEL
LIN {X 0,Y 204.412,Z 543.181,A -85,B 0,C 180,E1 -20974.388,E2 -20974.388} C_VEL
LIN {X 0,Y 204.681,Z 539.396,A -85,B 0,C 180,E1 -20977.895,E2 -20977.895} C_VEL
LIN {X 0,Y 205.239,Z 534.992,A -85,B 0,C 180,E1 -20980.856,E2 -20980.856} C_VEL
LIN {X 0,Y 206.14,Z 529.359,A -85,B 0,C 180,E1 -20983.808,E2 -20983.808} C_VEL
LIN {X 0,Y 207.665,Z 522.31,A -85,B 0,C 180,E1 -20986.719,E2 -20986.719} C_VEL
LIN {X 0,Y 209.208,Z 515.113,A -85,B 0,C 180,E1 -20989.12,E2 -20989.12} C_VEL
LIN {X 0,Y 210.652,Z 508.162,A -85,B 0,C 180,E1 -20991.057,E2 -20991.057} C_VEL
LIN {X 0,Y 212.8,Z 498.074,A -85,B 0,C 180,E1 -20993.349,E2 -20993.349} C_VEL
LIN {X 0,Y 213.363,Z 493.204,A -85,B 0,C 180,E1 -20994.315,E2 -20994.315} C_VEL
LIN {X 0,Y 212.829,Z 481.85,A -85,B 0,C 180,E1 -20996.373,E2 -20996.373} C_VEL
LIN {X 0,Y 211.815,Z 470.119,A -85,B 0,C 180,E1 -20998.14,E2 -20998.14} C_VEL
LIN {X 0,Y 210.208,Z 458.158,A -85,B 0,C 180,E1 -20999.625,E2 -20999.625} C_VEL
LIN {X 0,Y 207.742,Z 444.327,A -85,B 0,C 180,E1 -21001.006,E2 -21001.006} C_VEL
LIN {X 0,Y 207.165,Z 440.904,A -85,B 0,C 180,E1 -21001.335,E2 -21001.335} C_VEL
LIN {X 0,Y 208.235,Z 436.379,A -85,B 0,C 180,E1 -21005.903,E2 -21005.903} C_VEL
LIN {X 0,Y 208.293,Z 433.365,A -85,B 0,C 180,E1 -21009.1,E2 -21009.1} C_VEL
LIN {X 0,Y 207.744,Z 430.274,A -85,B 0,C 180,E1 -21012.579,E2 -21012.579} C_VEL
LIN {X 0,Y 207.045,Z 426.337,A -85,B 0,C 180,E1 -21017.243,E2 -21017.243} C_VEL
LIN {X 0,Y 206.744,Z 424.739,A -85,B 0,C 180,E1 -21019.406,E2 -21019.406} C_VEL
LIN {X 0,Y 206.701,Z 424.729,A -85,B 0,C 180,E1 -21024.689,E2 -21024.689} C_VEL
LIN {X 0,Y 206.725,Z 424.735,A -85,B 0,C 180,E1 -21029.339,E2 -21029.339} C_VEL
LIN {X 0,Y 206.735,Z 424.725,A -85,B 0,C 180,E1 -21033.772,E2 -21033.772} C_VEL
LIN {X 0,Y 206.76,Z 424.729,A -85,B 0,C 180,E1 -21038.043,E2 -21038.043} C_VEL
LIN {X 0,Y 206.876,Z 424.711,A -85,B 0,C 180,E1 -21042.197,E2 -21042.197} C_VEL
LIN {X 0,Y 206.916,Z 424.709,A -85,B 0,C 180,E1 -21046.246,E2 -21046.246} C_VEL
LIN {X 0,Y 207.108,Z 424.683,A -85,B 0,C 180,E1 -21050.231,E2 -21050.231} C_VEL
LIN {X 0,Y 207.17,Z 424.677,A -85,B 0,C 180,E1 -21052.201,E2 -21052.201} C_VEL
LIN {X 0,Y 207.384,Z 424.647,A -85,B 0,C 180,E1 -21058.058,E2 -21058.058} C_VEL
LIN {X 0,Y 207.513,Z 424.633,A -85,B 0,C 180,E1 -21060,E2 -21060} C_VEL
LIN {X 0,Y 207.384,Z 424.648,A -85,B 0,C 180,E1 -21061.942,E2 -21061.942} C_VEL
LIN {X 0,Y 207.17,Z 424.675,A -85,B 0,C 180,E1 -21067.799,E2 -21067.799} C_VEL
LIN {X 0,Y 206.984,Z 424.697,A -85,B 0,C 180,E1 -21071.755,E2 -21071.755} C_VEL
LIN {X 0,Y 206.869,Z 424.7,A -85,B 0,C 180,E1 -21075.77,E2 -21075.77} C_VEL
LIN {X 0,Y 206.786,Z 424.709,A -85,B 0,C 180,E1 -21079.869,E2 -21079.869} C_VEL
LIN {X 0,Y 206.766,Z 424.724,A -85,B 0,C 180,E1 -21084.072,E2 -21084.072} C_VEL
LIN {X 0,Y 206.746,Z 424.732,A -85,B 0,C 180,E1 -21088.418,E2 -21088.418} C_VEL
LIN {X 0,Y 206.704,Z 424.725,A -85,B 0,C 180,E1 -21092.957,E2 -21092.957} C_VEL
LIN {X 0,Y 206.681,Z 424.725,A -85,B 0,C 180,E1 -21097.74,E2 -21097.74} C_VEL
LIN {X 0,Y 206.642,Z 424.741,A -85,B 0,C 180,E1 -21101.562,E2 -21101.562} C_VEL
LIN {X 0,Y 206.632,Z 424.743,A -85,B 0,C 180,E1 -21105.582,E2 -21105.582} C_VEL
LIN {X 0,Y 206.667,Z 424.729,A -85,B 0,C 180,E1 -21109.749,E2 -21109.749} C_VEL
LIN {X 0,Y 206.733,Z 424.731,A -85,B 0,C 180,E1 -21114.695,E2 -21114.695} C_VEL
LIN {X 0,Y 206.725,Z 424.731,A -85,B 0,C 180,E1 -21119.339,E2 -21119.339} C_VEL
LIN {X 0,Y 206.735,Z 424.724,A -85,B 0,C 180,E1 -21123.772,E2 -21123.772} C_VEL
LIN {X 0,Y 206.76,Z 424.73,A -85,B 0,C 180,E1 -21128.043,E2 -21128.043} C_VEL
LIN {X 0,Y 206.876,Z 424.71,A -85,B 0,C 180,E1 -21132.196,E2 -21132.196} C_VEL
LIN {X 0,Y 206.916,Z 424.713,A -85,B 0,C 180,E1 -21136.245,E2 -21136.245} C_VEL
LIN {X 0,Y 207.135,Z 424.682,A -85,B 0,C 180,E1 -21140.232,E2 -21140.232} C_VEL
LIN {X 0,Y 207.191,Z 424.678,A -85,B 0,C 180,E1 -21142.201,E2 -21142.201} C_VEL
LIN {X 0,Y 207.384,Z 424.649,A -85,B 0,C 180,E1 -21148.057,E2 -21148.057} C_VEL
LIN {X 0,Y 207.516,Z 424.638,A -85,B 0,C 180,E1 -21149.999,E2 -21149.999} C_VEL
LIN {X 0,Y 207.374,Z 424.653,A -85,B 0,C 180,E1 -21151.941,E2 -21151.941} C_VEL
LIN {X 0,Y 206.83,Z 424.719,A -85,B 0,C 180,E1 -21157.811,E2 -21157.811} C_VEL
LIN {X 0,Y 206.552,Z 424.999,A -85,B 0,C 180,E1 -21159.343,E2 -21159.343} C_VEL
LIN {X 0,Y 206.224,Z 426.665,A -85,B 0,C 180,E1 -21161.673,E2 -21161.673} C_VEL
LIN {X 0,Y 210.162,Z 441.401,A -85,B 0,C 180,E1 -21163.315,E2 -21163.315} C_VEL
LIN {X 0,Y 212.78,Z 453.292,A -85,B 0,C 180,E1 -21164.892,E2 -21164.892} C_VEL
LIN {X 0,Y 214.65,Z 464.56,A -85,B 0,C 180,E1 -21166.647,E2 -21166.647} C_VEL
LIN {X 0,Y 215.573,Z 471.637,A -85,B 0,C 180,E1 -21167.918,E2 -21167.918} C_VEL
LIN {X 0,Y 213.614,Z 482.774,A -85,B 0,C 180,E1 -21169.958,E2 -21169.958} C_VEL
LIN {X 0,Y 211.425,Z 493.158,A -85,B 0,C 180,E1 -21172.36,E2 -21172.36} C_VEL
LIN {X 0,Y 209.414,Z 502.336,A -85,B 0,C 180,E1 -21175.024,E2 -21175.024} C_VEL
LIN {X 0,Y 207.817,Z 509.708,A -85,B 0,C 180,E1 -21177.687,E2 -21177.687} C_VEL
LIN {X 0,Y 206.403,Z 516.366,A -85,B 0,C 180,E1 -21180.713,E2 -21180.713} C_VEL
LIN {X 0,Y 205.339,Z 521.852,A -85,B 0,C 180,E1 -21183.921,E2 -21183.921} C_VEL
LIN {X 0,Y 204.68,Z 525.514,A -85,B 0,C 180,E1 -21186.709,E2 -21186.709} C_VEL
LIN {X 0,Y 204.251,Z 528.251,A -85,B 0,C 180,E1 -21189.492,E2 -21189.492} C_VEL
LIN {X 0,Y 204.135,Z 529.281,A -85,B 0,C 180,E1 -21190.853,E2 -21190.853} C_VEL
LIN {X 0,Y 204.048,Z 530.763,A -85,B 0,C 180,E1 -21193.672,E2 -21193.672} C_VEL
LIN {X 0,Y 204.282,Z 531.432,A -85,B 0,C 180,E1 -21196.523,E2 -21196.523} C_VEL
LIN {X 0,Y 204.823,Z 531.304,A -85,B 0,C 180,E1 -21199.312,E2 -21199.312} C_VEL
LIN {X 0,Y 205.684,Z 530.433,A -85,B 0,C 180,E1 -21202.045,E2 -21202.045} C_VEL
LIN {X 0,Y 207.508,Z 527.713,A -85,B 0,C 180,E1 -21206.025,E2 -21206.025} C_VEL
LIN {X 0,Y 210.032,Z 523.341,A -85,B 0,C 180,E1 -21209.873,E2 -21209.873} C_VEL
LIN {X 0,Y 212.808,Z 518.099,A -85,B 0,C 180,E1 -21213.082,E2 -21213.082} C_VEL
LIN {X 0,Y 215.743,Z 512.29,A -85,B 0,C 180,E1 -21215.798,E2 -21215.798} C_VEL
LIN {X 0,Y 219.143,Z 505.116,A -85,B 0,C 180,E1 -21218.438,E2 -21218.438} C_VEL
LIN {X 0,Y 222.997,Z 496.197,A -85,B 0,C 180,E1 -21220.99,E2 -21220.99} C_VEL
LIN {X 0,Y 226.682,Z 486.52,A -85,B 0,C 180,E1 -21223.172,E2 -21223.172} C_VEL
LIN {X 0,Y 226.931,Z 482.214,A -85,B 0,C 180,E1 -21224.277,E2 -21224.277} C_VEL
LIN {X 0,Y 226.301,Z 473.679,A -85,B 0,C 180,E1 -21226.531,E2 -21226.531} C_VEL
LIN {X 0,Y 224.715,Z 464.908,A -85,B 0,C 180,E1 -21228.849,E2 -21228.849} C_VEL
LIN {X 0,Y 222.168,Z 456.051,A -85,B 0,C 180,E1 -21231.309,E2 -21231.309} C_VEL
LIN {X 0,Y 219.787,Z 450.051,A -85,B 0,C 180,E1 -21233.113,E2 -21233.113} C_VEL
LIN {X 0,Y 217.859,Z 446.111,A -85,B 0,C 180,E1 -21234.446,E2 -21234.446} C_VEL
LIN {X 0,Y 214.589,Z 440.736,A -85,B 0,C 180,E1 -21236.538,E2 -21236.538} C_VEL
LIN {X 0,Y 212.604,Z 437.487,A -85,B 0,C 180,E1 -21237.869,E2 -21237.869} C_VEL
LIN {X 0,Y 211.946,Z 436.077,A -85,B 0,C 180,E1 -21238.362,E2 -21238.362} C_VEL
LIN {X 0,Y 209.701,Z 433.543,A -85,B 0,C 180,E1 -21239.784,E2 -21239.784} C_VEL
LIN {X 0,Y 208.486,Z 430.724,A -85,B 0,C 180,E1 -21240.845,E2 -21240.845} C_VEL
LIN {X 0,Y 208.025,Z 429.782,A -85,B 0,C 180,E1 -21245.817,E2 -21245.817} C_VEL
LIN {X 0,Y 207.924,Z 429.291,A -85,B 0,C 180,E1 -21249.73,E2 -21249.73} C_VEL
LIN {X 0,Y 207.684,Z 429.129,A -85,B 0,C 180,E1 -21253.703,E2 -21253.703} C_VEL
LIN {X 0,Y 207.703,Z 429.222,A -85,B 0,C 180,E1 -21257.73,E2 -21257.73} C_VEL
LIN {X 0,Y 207.707,Z 429.671,A -85,B 0,C 180,E1 -21261.851,E2 -21261.851} C_VEL
LIN {X 0,Y 207.805,Z 430.486,A -85,B 0,C 180,E1 -21266.083,E2 -21266.083} C_VEL
LIN {X 0,Y 207.965,Z 431.721,A -85,B 0,C 180,E1 -21270.459,E2 -21270.459} C_VEL
LIN {X 0,Y 208.249,Z 433.415,A -85,B 0,C 180,E1 -21275.01,E2 -21275.01} C_VEL
LIN {X 0,Y 208.64,Z 435.638,A -85,B 0,C 180,E1 -21279.793,E2 -21279.793} C_VEL
LIN {X 0,Y 208.912,Z 437.248,A -85,B 0,C 180,E1 -21282.449,E2 -21282.449} C_VEL
LIN {X 0,Y 210.09,Z 440.238,A -85,B 0,C 180,E1 -21283.379,E2 -21283.379} C_VEL
LIN {X 0,Y 212.803,Z 443.814,A -85,B 0,C 180,E1 -21285.074,E2 -21285.074} C_VEL
LIN {X 0,Y 214.599,Z 447.643,A -85,B 0,C 180,E1 -21286.305,E2 -21286.305} C_VEL
LIN {X 0,Y 215.965,Z 449.746,A -85,B 0,C 180,E1 -21287.116,E2 -21287.116} C_VEL
LIN {X 0,Y 218.774,Z 455.964,A -85,B 0,C 180,E1 -21289.019,E2 -21289.019} C_VEL
LIN {X 0,Y 221.081,Z 462.349,A -85,B 0,C 180,E1 -21290.743,E2 -21290.743} C_VEL
LIN {X 0,Y 222.916,Z 470.857,A -85,B 0,C 180,E1 -21292.757,E2 -21292.757} C_VEL
LIN {X 0,Y 224.196,Z 481.705,A -85,B 0,C 180,E1 -21295.2,E2 -21295.2} C_VEL
LIN {X 0,Y 224.272,Z 492.022,A -85,B 0,C 180,E1 -21297.559,E2 -21297.559} C_VEL
LIN {X 0,Y 223.298,Z 501.297,A -85,B 0,C 180,E1 -21299.764,E2 -21299.764} C_VEL
LIN {X 0,Y 222.063,Z 506.8,A -85,B 0,C 180,E1 -21301.143,E2 -21301.143} C_VEL
LIN {X 0,Y 217.949,Z 516.424,A -85,B 0,C 180,E1 -21303.681,E2 -21303.681} C_VEL
LIN {X 0,Y 217.207,Z 518.115,A -85,B 0,C 180,E1 -21304.195,E2 -21304.195} C_VEL
LIN {X 0,Y 215.038,Z 521.732,A -85,B 0,C 180,E1 -21305.316,E2 -21305.316} C_VEL
LIN {X 0,Y 207.909,Z 529.229,A -85,B 0,C 180,E1 -21307.824,E2 -21307.824} C_VEL
LIN {X 0,Y 204.332,Z 532.932,A -85,B 0,C 180,E1 -21309.479,E2 -21309.479} C_VEL
LIN {X 0,Y 203.185,Z 534.579,A -85,B 0,C 180,E1 -21310.417,E2 -21310.417} C_VEL
LIN {X 0,Y 200.583,Z 539.316,A -85,B 0,C 180,E1 -21313.723,E2 -21313.723} C_VEL
LIN {X 0,Y 199.446,Z 541.504,A -85,B 0,C 180,E1 -21315.721,E2 -21315.721} C_VEL
LIN {X 0,Y 198.025,Z 544.619,A -85,B 0,C 180,E1 -21319.779,E2 -21319.779} C_VEL
LIN {X 0,Y 197.339,Z 546.191,A -85,B 0,C 180,E1 -21323.868,E2 -21323.868} C_VEL
LIN {X 0,Y 197.376,Z 546.157,A -85,B 0,C 180,E1 -21327.96,E2 -21327.96} C_VEL
LIN {X 0,Y 197.533,Z 545.561,A -85,B 0,C 180,E1 -21330.001,E2 -21330.001} C_VEL
LIN {X 0,Y 197.415,Z 544.543,A -85,B 0,C 180,E1 -21332.041,E2 -21332.041} C_VEL
LIN {X 0,Y 197.344,Z 542.857,A -85,B 0,C 180,E1 -21334.315,E2 -21334.315} C_VEL
LIN {X 0,Y 197.644,Z 538.776,A -85,B 0,C 180,E1 -21338.178,E2 -21338.178} C_VEL
LIN {X 0,Y 198.222,Z 534.265,A -85,B 0,C 180,E1 -21341.246,E2 -21341.246} C_VEL
LIN {X 0,Y 199.473,Z 527.385,A -85,B 0,C 180,E1 -21344.8,E2 -21344.8} C_VEL
LIN {X 0,Y 201.059,Z 519.911,A -85,B 0,C 180,E1 -21347.81,E2 -21347.81} C_VEL
LIN {X 0,Y 202.396,Z 513.921,A -85,B 0,C 180,E1 -21349.79,E2 -21349.79} C_VEL
LIN {X 0,Y 204.402,Z 505.048,A -85,B 0,C 180,E1 -21352.224,E2 -21352.224} C_VEL
LIN {X 0,Y 206.433,Z 495.335,A -85,B 0,C 180,E1 -21354.381,E2 -21354.381} C_VEL
LIN {X 0,Y 206.032,Z 484.148,A -85,B 0,C 180,E1 -21356.571,E2 -21356.571} C_VEL
LIN {X 0,Y 205.168,Z 472.562,A -85,B 0,C 180,E1 -21358.451,E2 -21358.451} C_VEL
LIN {X 0,Y 203.657,Z 460.147,A -85,B 0,C 180,E1 -21360.13,E2 -21360.13} C_VEL
LIN {X 0,Y 201.467,Z 447.152,A -85,B 0,C 180,E1 -21361.552,E2 -21361.552} C_VEL
LIN {X 0,Y 200.248,Z 440.674,A -85,B 0,C 180,E1 -21362.136,E2 -21362.136} C_VEL
LIN {X 0,Y 201.214,Z 436.615,A -85,B 0,C 180,E1 -21366.426,E2 -21366.426} C_VEL
LIN {X 0,Y 201.178,Z 433.588,A -85,B 0,C 180,E1 -21369.775,E2 -21369.775} C_VEL
LIN {X 0,Y 200.402,Z 429.566,A -85,B 0,C 180,E1 -21374.539,E2 -21374.539} C_VEL
LIN {X 0,Y 199.705,Z 425.639,A -85,B 0,C 180,E1 -21379.462,E2 -21379.462} C_VEL
LIN {X 0,Y 199.618,Z 425.61,A -85,B 0,C 180,E1 -21384.074,E2 -21384.074} C_VEL
LIN {X 0,Y 199.703,Z 425.609,A -85,B 0,C 180,E1 -21388.137,E2 -21388.137} C_VEL
LIN {X 0,Y 199.689,Z 425.6,A -85,B 0,C 180,E1 -21392.772,E2 -21392.772} C_VEL
LIN {X 0,Y 199.74,Z 425.606,A -85,B 0,C 180,E1 -21397.229,E2 -21397.229} C_VEL
LIN {X 0,Y 199.799,Z 425.593,A -85,B 0,C 180,E1 -21401.758,E2 -21401.758} C_VEL
LIN {X 0,Y 199.85,Z 425.589,A -85,B 0,C 180,E1 -21405.749,E2 -21405.749} C_VEL
LIN {X 0,Y 200.073,Z 425.559,A -85,B 0,C 180,E1 -21409.884,E2 -21409.884} C_VEL
LIN {X 0,Y 200.037,Z 425.564,A -85,B 0,C 180,E1 -21413.95,E2 -21413.95} C_VEL
LIN {X 0,Y 200.323,Z 425.526,A -85,B 0,C 180,E1 -21417.989,E2 -21417.989} C_VEL
LIN {X 0,Y 200.478,Z 425.509,A -85,B 0,C 180,E1 -21420,E2 -21420} C_VEL
LIN {X 0,Y 200.032,Z 425.561,A -85,B 0,C 180,E1 -21424.029,E2 -21424.029} C_VEL
LIN {X 0,Y 200.114,Z 425.554,A -85,B 0,C 180,E1 -21428.076,E2 -21428.076} C_VEL
LIN {X 0,Y 199.916,Z 425.577,A -85,B 0,C 180,E1 -21432.177,E2 -21432.177} C_VEL
LIN {X 0,Y 199.806,Z 425.577,A -85,B 0,C 180,E1 -21436.343,E2 -21436.343} C_VEL
LIN {X 0,Y 199.702,Z 425.593,A -85,B 0,C 180,E1 -21440.605,E2 -21440.605} C_VEL
LIN {X 0,Y 199.675,Z 425.613,A -85,B 0,C 180,E1 -21444.984,E2 -21444.984} C_VEL
LIN {X 0,Y 199.677,Z 425.609,A -85,B 0,C 180,E1 -21449.522,E2 -21449.522} C_VEL
LIN {X 0,Y 199.679,Z 425.604,A -85,B 0,C 180,E1 -21452.358,E2 -21452.358} C_VEL
LIN {X 0,Y 199.624,Z 425.598,A -85,B 0,C 180,E1 -21456.763,E2 -21456.763} C_VEL
LIN {X 0,Y 199.609,Z 425.613,A -85,B 0,C 180,E1 -21459.328,E2 -21459.328} C_VEL
LIN {X 0,Y 199.574,Z 425.623,A -85,B 0,C 180,E1 -21462.309,E2 -21462.309} C_VEL
LIN {X 0,Y 199.578,Z 425.622,A -85,B 0,C 180,E1 -21465.228,E2 -21465.228} C_VEL
LIN {X 0,Y 199.64,Z 425.601,A -85,B 0,C 180,E1 -21470.679,E2 -21470.679} C_VEL
LIN {X 0,Y 199.637,Z 425.614,A -85,B 0,C 180,E1 -21475.718,E2 -21475.718} C_VEL
LIN {X 0,Y 199.706,Z 425.609,A -85,B 0,C 180,E1 -21478.137,E2 -21478.137} C_VEL
LIN {X 0,Y 199.689,Z 425.601,A -85,B 0,C 180,E1 -21482.771,E2 -21482.771} C_VEL
LIN {X 0,Y 199.741,Z 425.603,A -85,B 0,C 180,E1 -21487.229,E2 -21487.229} C_VEL
LIN {X 0,Y 199.799,Z 425.59,A -85,B 0,C 180,E1 -21491.757,E2 -21491.757} C_VEL
LIN {X 0,Y 199.85,Z 425.591,A -85,B 0,C 180,E1 -21495.749,E2 -21495.749} C_VEL
LIN {X 0,Y 200.078,Z 425.559,A -85,B 0,C 180,E1 -21499.884,E2 -21499.884} C_VEL
LIN {X 0,Y 200.135,Z 425.556,A -85,B 0,C 180,E1 -21501.925,E2 -21501.925} C_VEL
LIN {X 0,Y 200.323,Z 425.528,A -85,B 0,C 180,E1 -21507.989,E2 -21507.989} C_VEL
LIN {X 0,Y 200.48,Z 425.515,A -85,B 0,C 180,E1 -21509.999,E2 -21509.999} C_VEL
LIN {X 0,Y 200.311,Z 425.532,A -85,B 0,C 180,E1 -21512.01,E2 -21512.01} C_VEL
LIN {X 0,Y 199.88,Z 425.592,A -85,B 0,C 180,E1 -21516.054,E2 -21516.054} C_VEL
LIN {X 0,Y 199.558,Z 425.696,A -85,B 0,C 180,E1 -21519.057,E2 -21519.057} C_VEL
LIN {X 0,Y 199.267,Z 426.941,A -85,B 0,C 180,E1 -21520.862,E2 -21520.862} C_VEL
LIN {X 0,Y 202.673,Z 439.252,A -85,B 0,C 180,E1 -21522.23,E2 -21522.23} C_VEL
LIN {X 0,Y 205.436,Z 451.373,A -85,B 0,C 180,E1 -21523.854,E2 -21523.854} C_VEL
LIN {X 0,Y 207.464,Z 463.205,A -85,B 0,C 180,E1 -21525.723,E2 -21525.723} C_VEL
LIN {X 0,Y 208.673,Z 472.256,A -85,B 0,C 180,E1 -21527.391,E2 -21527.391} C_VEL
LIN {X 0,Y 207.448,Z 479.815,A -85,B 0,C 180,E1 -21528.787,E2 -21528.787} C_VEL
LIN {X 0,Y 205.27,Z 490.115,A -85,B 0,C 180,E1 -21531.068,E2 -21531.068} C_VEL
LIN {X 0,Y 203.306,Z 498.713,A -85,B 0,C 180,E1 -21533.423,E2 -21533.423} C_VEL
LIN {X 0,Y 201.3,Z 507.791,A -85,B 0,C 180,E1 -21536.549,E2 -21536.549} C_VEL
LIN {X 0,Y 199.751,Z 514.583,A -85,B 0,C 180,E1 -21539.509,E2 -21539.509} C_VEL
LIN {X 0,Y 198.592,Z 520.296,A -85,B 0,C 180,E1 -21542.661,E2 -21542.661} C_VEL
LIN {X 0,Y 197.705,Z 525.125,A -85,B 0,C 180,E1 -21546.151,E2 -21546.151} C_VEL
LIN {X 0,Y 197.103,Z 528.739,A -85,B 0,C 180,E1 -21549.926,E2 -21549.926} C_VEL
LIN {X 0,Y 196.962,Z 530.492,A -85,B 0,C 180,E1 -21552.683,E2 -21552.683} C_VEL
LIN {X 0,Y 197.054,Z 531.494,A -85,B 0,C 180,E1 -21555.503,E2 -21555.503} C_VEL
LIN {X 0,Y 197.502,Z 531.755,A -85,B 0,C 180,E1 -21558.353,E2 -21558.353} C_VEL
LIN {X 0,Y 198.283,Z 531.261,A -85,B 0,C 180,E1 -21561.238,E2 -21561.238} C_VEL
LIN {X 0,Y 199.419,Z 529.96,A -85,B 0,C 180,E1 -21564.15,E2 -21564.15} C_VEL
LIN {X 0,Y 200.96,Z 527.766,A -85,B 0,C 180,E1 -21567.068,E2 -21567.068} C_VEL
LIN {X 0,Y 202.914,Z 524.638,A -85,B 0,C 180,E1 -21569.981,E2 -21569.981} C_VEL
LIN {X 0,Y 205.347,Z 520.507,A -85,B 0,C 180,E1 -21572.852,E2 -21572.852} C_VEL
LIN {X 0,Y 208.242,Z 515.239,A -85,B 0,C 180,E1 -21575.673,E2 -21575.673} C_VEL
LIN {X 0,Y 211.993,Z 508.094,A -85,B 0,C 180,E1 -21578.613,E2 -21578.613} C_VEL
LIN {X 0,Y 215.522,Z 500.609,A -85,B 0,C 180,E1 -21581.023,E2 -21581.023} C_VEL
LIN {X 0,Y 219.802,Z 490.518,A -85,B 0,C 180,E1 -21583.578,E2 -21583.578} C_VEL
LIN {X 0,Y 220.876,Z 487.587,A -85,B 0,C 180,E1 -21584.221,E2 -21584.221} C_VEL
LIN {X 0,Y 220.835,Z 478.982,A -85,B 0,C 180,E1 -21586.66,E2 -21586.66} C_VEL
LIN {X 0,Y 219.834,Z 470.928,A -85,B 0,C 180,E1 -21588.941,E2 -21588.941} C_VEL
LIN {X 0,Y 217.825,Z 462.099,A -85,B 0,C 180,E1 -21591.552,E2 -21591.552} C_VEL
LIN {X 0,Y 215.693,Z 455.693,A -85,B 0,C 180,E1 -21593.57,E2 -21593.57} C_VEL
LIN {X 0,Y 213.107,Z 450.309,A -85,B 0,C 180,E1 -21595.588,E2 -21595.588} C_VEL
LIN {X 0,Y 211.107,Z 446.581,A -85,B 0,C 180,E1 -21597.097,E2 -21597.097} C_VEL
LIN {X 0,Y 209.402,Z 443.711,A -85,B 0,C 180,E1 -21598.396,E2 -21598.396} C_VEL
LIN {X 0,Y 208.431,Z 441.801,A -85,B 0,C 180,E1 -21599.195,E2 -21599.195} C_VEL
LIN {X 0,Y 206.382,Z 438.86,A -85,B 0,C 180,E1 -21600.732,E2 -21600.732} C_VEL
LIN {X 0,Y 205.609,Z 437.118,A -85,B 0,C 180,E1 -21601.469,E2 -21601.469} C_VEL
LIN {X 0,Y 202.631,Z 434.644,A -85,B 0,C 180,E1 -21603.704,E2 -21603.704} C_VEL
LIN {X 0,Y 201.227,Z 431.926,A -85,B 0,C 180,E1 -21605.135,E2 -21605.135} C_VEL
LIN {X 0,Y 201.141,Z 431.484,A -85,B 0,C 180,E1 -21605.388,E2 -21605.388} C_VEL
LIN {X 0,Y 201.009,Z 430.947,A -85,B 0,C 180,E1 -21610.068,E2 -21610.068} C_VEL
LIN {X 0,Y 200.787,Z 430.866,A -85,B 0,C 180,E1 -21616.261,E2 -21616.261} C_VEL
LIN {X 0,Y 200.76,Z 431.214,A -85,B 0,C 180,E1 -21620.492,E2 -21620.492} C_VEL
LIN {X 0,Y 200.854,Z 431.914,A -85,B 0,C 180,E1 -21624.828,E2 -21624.828} C_VEL
LIN {X 0,Y 201.019,Z 433.03,A -85,B 0,C 180,E1 -21629.306,E2 -21629.306} C_VEL
LIN {X 0,Y 201.239,Z 434.623,A -85,B 0,C 180,E1 -21633.972,E2 -21633.972} C_VEL
LIN {X 0,Y 201.542,Z 436.343,A -85,B 0,C 180,E1 -21638.006,E2 -21638.006} C_VEL
LIN {X 0,Y 202.583,Z 439.059,A -85,B 0,C 180,E1 -21639.083,E2 -21639.083} C_VEL
LIN {X 0,Y 204.939,Z 442.373,A -85,B 0,C 180,E1 -21641.025,E2 -21641.025} C_VEL
LIN {X 0,Y 205.927,Z 443.48,A -85,B 0,C 180,E1 -21641.73,E2 -21641.73} C_VEL
LIN {X 0,Y 207.568,Z 447.089,A -85,B 0,C 180,E1 -21643.118,E2 -21643.118} C_VEL
LIN {X 0,Y 209.172,Z 449.143,A -85,B 0,C 180,E1 -21644.199,E2 -21644.199} C_VEL
LIN {X 0,Y 210.846,Z 453.046,A -85,B 0,C 180,E1 -21645.576,E2 -21645.576} C_VEL
LIN {X 0,Y 211.7,Z 454.286,A -85,B 0,C 180,E1 -21646.123,E2 -21646.123} C_VEL
LIN {X 0,Y 214.584,Z 461.19,A -85,B 0,C 180,E1 -21648.393,E2 -21648.393} C_VEL
LIN {X 0,Y 216.155,Z 466.092,A -85,B 0,C 180,E1 -21649.823,E2 -21649.823} C_VEL
LIN {X 0,Y 217.687,Z 474.449,A -85,B 0,C 180,E1 -21651.938,E2 -21651.938} C_VEL
LIN {X 0,Y 218.534,Z 485.542,A -85,B 0,C 180,E1 -21654.63,E2 -21654.63} C_VEL
LIN {X 0,Y 218.239,Z 494.645,A -85,B 0,C 180,E1 -21656.855,E2 -21656.855} C_VEL
LIN {X 0,Y 216.858,Z 504.159,A -85,B 0,C 180,E1 -21659.309,E2 -21659.309} C_VEL
LIN {X 0,Y 215.914,Z 507.684,A -85,B 0,C 180,E1 -21660.24,E2 -21660.24} C_VEL
LIN {X 0,Y 211.648,Z 517.122,A -85,B 0,C 180,E1 -21662.834,E2 -21662.834} C_VEL
LIN {X 0,Y 207.974,Z 524.746,A -85,B 0,C 180,E1 -21665.547,E2 -21665.547} C_VEL
LIN {X 0,Y 204.572,Z 531.84,A -85,B 0,C 180,E1 -21668.856,E2 -21668.856} C_VEL
LIN {X 0,Y 203.185,Z 534.579,A -85,B 0,C 180,E1 -21670.417,E2 -21670.417} C_VEL
LIN {X 0,Y 201.329,Z 536.933,A -85,B 0,C 180,E1 -21671.861,E2 -21671.861} C_VEL
LIN {X 0,Y 196.779,Z 540.212,A -85,B 0,C 180,E1 -21674.217,E2 -21674.217} C_VEL
LIN {X 0,Y 192.568,Z 542.774,A -85,B 0,C 180,E1 -21676.748,E2 -21676.748} C_VEL
LIN {X 0,Y 191.285,Z 543.907,A -85,B 0,C 180,E1 -21678.429,E2 -21678.429} C_VEL
LIN {X 0,Y 190.531,Z 545.434,A -85,B 0,C 180,E1 -21681.516,E2 -21681.516} C_VEL
LIN {X 0,Y 190.164,Z 546.06,A -85,B 0,C 180,E1 -21685.762,E2 -21685.762} C_VEL
LIN {X 0,Y 190.274,Z 545.806,A -85,B 0,C 180,E1 -21687.884,E2 -21687.884} C_VEL
LIN {X 0,Y 190.447,Z 545.165,A -85,B 0,C 180,E1 -21690.001,E2 -21690.001} C_VEL
LIN {X 0,Y 190.334,Z 544.062,A -85,B 0,C 180,E1 -21692.117,E2 -21692.117} C_VEL
LIN {X 0,Y 190.277,Z 542.523,A -85,B 0,C 180,E1 -21694.237,E2 -21694.237} C_VEL
LIN {X 0,Y 190.466,Z 539.391,A -85,B 0,C 180,E1 -21697.421,E2 -21697.421} C_VEL
LIN {X 0,Y 190.986,Z 535.162,A -85,B 0,C 180,E1 -21700.603,E2 -21700.603} C_VEL
LIN {X 0,Y 192.073,Z 528.696,A -85,B 0,C 180,E1 -21704.3,E2 -21704.3} C_VEL
LIN {X 0,Y 193.7,Z 521.606,A -85,B 0,C 180,E1 -21707.418,E2 -21707.418} C_VEL
LIN {X 0,Y 195.328,Z 514.372,A -85,B 0,C 180,E1 -21709.988,E2 -21709.988} C_VEL
LIN {X 0,Y 197.145,Z 506.503,A -85,B 0,C 180,E1 -21712.287,E2 -21712.287} C_VEL
LIN {X 0,Y 199.443,Z 496.093,A -85,B 0,C 180,E1 -21714.738,E2 -21714.738} C_VEL
LIN {X 0,Y 199.178,Z 485.079,A -85,B 0,C 180,E1 -21717.02,E2 -21717.02} C_VEL
LIN {X 0,Y 198.445,Z 474.141,A -85,B 0,C 180,E1 -21718.909,E2 -21718.909} C_VEL
LIN {X 0,Y 197.135,Z 462.582,A -85,B 0,C 180,E1 -21720.576,E2 -21720.576} C_VEL
LIN {X 0,Y 194.928,Z 448.69,A -85,B 0,C 180,E1 -21722.217,E2 -21722.217} C_VEL
LIN {X 0,Y 193.356,Z 440.417,A -85,B 0,C 180,E1 -21723.04,E2 -21723.04} C_VEL
LIN {X 0,Y 193.975,Z 438.211,A -85,B 0,C 180,E1 -21725.43,E2 -21725.43} C_VEL
LIN {X 0,Y 194.214,Z 435.961,A -85,B 0,C 180,E1 -21727.966,E2 -21727.966} C_VEL
LIN {X 0,Y 193.745,Z 432.525,A -85,B 0,C 180,E1 -21732.046,E2 -21732.046} C_VEL
LIN {X 0,Y 193.048,Z 428.798,A -85,B 0,C 180,E1 -21736.729,E2 -21736.729} C_VEL
LIN {X 0,Y 192.643,Z 426.495,A -85,B 0,C 180,E1 -21740.008,E2 -21740.008} C_VEL
LIN {X 0,Y 192.564,Z 426.488,A -85,B 0,C 180,E1 -21744.271,E2 -21744.271} C_VEL
LIN {X 0,Y 192.613,Z 426.494,A -85,B 0,C 180,E1 -21747.058,E2 -21747.058} C_VEL
LIN {X 0,Y 192.667,Z 426.477,A -85,B 0,C 180,E1 -21751.692,E2 -21751.692} C_VEL
LIN {X 0,Y 192.708,Z 426.477,A -85,B 0,C 180,E1 -21756.349,E2 -21756.349} C_VEL
LIN {X 0,Y 192.734,Z 426.473,A -85,B 0,C 180,E1 -21761.458,E2 -21761.458} C_VEL
LIN {X 0,Y 192.774,Z 426.473,A -85,B 0,C 180,E1 -21765.214,E2 -21765.214} C_VEL
LIN {X 0,Y 192.984,Z 426.443,A -85,B 0,C 180,E1 -21769.508,E2 -21769.508} C_VEL
LIN {X 0,Y 193.065,Z 426.434,A -85,B 0,C 180,E1 -21771.627,E2 -21771.627} C_VEL
LIN {X 0,Y 193.265,Z 426.406,A -85,B 0,C 180,E1 -21777.916,E2 -21777.916} C_VEL
LIN {X 0,Y 193.443,Z 426.386,A -85,B 0,C 180,E1 -21780,E2 -21780} C_VEL
LIN {X 0,Y 192.978,Z 426.44,A -85,B 0,C 180,E1 -21784.177,E2 -21784.177} C_VEL
LIN {X 0,Y 193.064,Z 426.433,A -85,B 0,C 180,E1 -21788.372,E2 -21788.372} C_VEL
LIN {X 0,Y 192.855,Z 426.457,A -85,B 0,C 180,E1 -21792.63,E2 -21792.63} C_VEL
LIN {X 0,Y 192.76,Z 426.448,A -85,B 0,C 180,E1 -21796.958,E2 -21796.958} C_VEL
LIN {X 0,Y 192.639,Z 426.478,A -85,B 0,C 180,E1 -21801.397,E2 -21801.397} C_VEL
LIN {X 0,Y 192.666,Z 426.481,A -85,B 0,C 180,E1 -21804.224,E2 -21804.224} C_VEL
LIN {X 0,Y 192.652,Z 426.486,A -85,B 0,C 180,E1 -21808.892,E2 -21808.892} C_VEL
LIN {X 0,Y 192.601,Z 426.479,A -85,B 0,C 180,E1 -21813.185,E2 -21813.185} C_VEL
LIN {X 0,Y 192.553,Z 426.485,A -85,B 0,C 180,E1 -21818.352,E2 -21818.352} C_VEL
LIN {X 0,Y 192.491,Z 426.506,A -85,B 0,C 180,E1 -21823.095,E2 -21823.095} C_VEL
LIN {X 0,Y 192.492,Z 426.502,A -85,B 0,C 180,E1 -21826.904,E2 -21826.904} C_VEL
LIN {X 0,Y 192.576,Z 426.48,A -85,B 0,C 180,E1 -21831.653,E2 -21831.653} C_VEL
LIN {X 0,Y 192.6,Z 426.488,A -85,B 0,C 180,E1 -21834.278,E2 -21834.278} C_VEL
LIN {X 0,Y 192.61,Z 426.49,A -85,B 0,C 180,E1 -21839.28,E2 -21839.28} C_VEL
LIN {X 0,Y 192.667,Z 426.478,A -85,B 0,C 180,E1 -21841.692,E2 -21841.692} C_VEL
LIN {X 0,Y 192.708,Z 426.479,A -85,B 0,C 180,E1 -21846.348,E2 -21846.348} C_VEL
LIN {X 0,Y 192.734,Z 426.47,A -85,B 0,C 180,E1 -21851.457,E2 -21851.457} C_VEL
LIN {X 0,Y 192.774,Z 426.473,A -85,B 0,C 180,E1 -21855.214,E2 -21855.214} C_VEL
LIN {X 0,Y 193.022,Z 426.437,A -85,B 0,C 180,E1 -21859.51,E2 -21859.51} C_VEL
LIN {X 0,Y 193.006,Z 426.441,A -85,B 0,C 180,E1 -21863.728,E2 -21863.728} C_VEL
LIN {X 0,Y 193.265,Z 426.407,A -85,B 0,C 180,E1 -21867.915,E2 -21867.915} C_VEL
LIN {X 0,Y 193.444,Z 426.392,A -85,B 0,C 180,E1 -21869.999,E2 -21869.999} C_VEL
LIN {X 0,Y 192.915,Z 426.453,A -85,B 0,C 180,E1 -21874.178,E2 -21874.178} C_VEL
LIN {X 0,Y 192.656,Z 426.484,A -85,B 0,C 180,E1 -21878.39,E2 -21878.39} C_VEL
LIN {X 0,Y 192.393,Z 426.894,A -85,B 0,C 180,E1 -21879.497,E2 -21879.497} C_VEL
LIN {X 0,Y 192.353,Z 427.383,A -85,B 0,C 180,E1 -21879.983,E2 -21879.983} C_VEL
LIN {X 0,Y 195.693,Z 439.476,A -85,B 0,C 180,E1 -21881.391,E2 -21881.391} C_VEL
LIN {X 0,Y 198.318,Z 450.751,A -85,B 0,C 180,E1 -21882.958,E2 -21882.958} C_VEL
LIN {X 0,Y 200.311,Z 461.777,A -85,B 0,C 180,E1 -21884.735,E2 -21884.735} C_VEL
LIN {X 0,Y 201.755,Z 472.229,A -85,B 0,C 180,E1 -21886.7,E2 -21886.7} C_VEL
LIN {X 0,Y 201.707,Z 474.963,A -85,B 0,C 180,E1 -21887.226,E2 -21887.226} C_VEL
LIN {X 0,Y 199.246,Z 486.515,A -85,B 0,C 180,E1 -21889.618,E2 -21889.618} C_VEL
LIN {X 0,Y 197.147,Z 495.838,A -85,B 0,C 180,E1 -21892.049,E2 -21892.049} C_VEL
LIN {X 0,Y 195.036,Z 504.788,A -85,B 0,C 180,E1 -21894.981,E2 -21894.981} C_VEL
LIN {X 0,Y 193.191,Z 512.627,A -85,B 0,C 180,E1 -21898.223,E2 -21898.223} C_VEL
LIN {X 0,Y 191.809,Z 519.058,A -85,B 0,C 180,E1 -21901.621,E2 -21901.621} C_VEL
LIN {X 0,Y 190.921,Z 523.488,A -85,B 0,C 180,E1 -21904.63,E2 -21904.63} C_VEL
LIN {X 0,Y 190.301,Z 526.794,A -85,B 0,C 180,E1 -21907.542,E2 -21907.542} C_VEL
LIN {X 0,Y 190.101,Z 528.186,A -85,B 0,C 180,E1 -21909.071,E2 -21909.071} C_VEL
LIN {X 0,Y 189.869,Z 530.37,A -85,B 0,C 180,E1 -21912.243,E2 -21912.243} C_VEL
LIN {X 0,Y 189.936,Z 531.628,A -85,B 0,C 180,E1 -21915.329,E2 -21915.329} C_VEL
LIN {X 0,Y 190.397,Z 532.066,A -85,B 0,C 180,E1 -21918.362,E2 -21918.362} C_VEL
LIN {X 0,Y 191.189,Z 531.714,A -85,B 0,C 180,E1 -21921.324,E2 -21921.324} C_VEL
LIN {X 0,Y 192.304,Z 530.594,A -85,B 0,C 180,E1 -21924.215,E2 -21924.215} C_VEL
LIN {X 0,Y 193.782,Z 528.772,A -85,B 0,C 180,E1 -21927.043,E2 -21927.043} C_VEL
LIN {X 0,Y 195.575,Z 526.246,A -85,B 0,C 180,E1 -21929.795,E2 -21929.795} C_VEL
LIN {X 0,Y 197.862,Z 522.719,A -85,B 0,C 180,E1 -21932.619,E2 -21932.619} C_VEL
LIN {X 0,Y 201.339,Z 516.932,A -85,B 0,C 180,E1 -21936.072,E2 -21936.072} C_VEL
LIN {X 0,Y 205.391,Z 509.799,A -85,B 0,C 180,E1 -21939.229,E2 -21939.229} C_VEL
LIN {X 0,Y 209.748,Z 501.253,A -85,B 0,C 180,E1 -21942.139,E2 -21942.139} C_VEL
LIN {X 0,Y 213.837,Z 492.217,A -85,B 0,C 180,E1 -21944.516,E2 -21944.516} C_VEL
LIN {X 0,Y 214.884,Z 489.778,A -85,B 0,C 180,E1 -21945.075,E2 -21945.075} C_VEL
LIN {X 0,Y 215.11,Z 482.495,A -85,B 0,C 180,E1 -21947.26,E2 -21947.26} C_VEL
LIN {X 0,Y 214.476,Z 474.782,A -85,B 0,C 180,E1 -21949.616,E2 -21949.616} C_VEL
LIN {X 0,Y 212.586,Z 465.228,A -85,B 0,C 180,E1 -21952.643,E2 -21952.643} C_VEL
LIN {X 0,Y 211.191,Z 460.514,A -85,B 0,C 180,E1 -21954.271,E2 -21954.271} C_VEL
LIN {X 0,Y 208.146,Z 453.663,A -85,B 0,C 180,E1 -21957.056,E2 -21957.056} C_VEL
LIN {X 0,Y 204.806,Z 447.433,A -85,B 0,C 180,E1 -21960,E2 -21960} C_VEL
LIN {X 0,Y 203.101,Z 444.319,A -85,B 0,C 180,E1 -21961.611,E2 -21961.611} C_VEL
LIN {X 0,Y 202.567,Z 443.349,A -85,B 0,C 180,E1 -21962.144,E2 -21962.144} C_VEL
LIN {X 0,Y 199.898,Z 440.704,A -85,B 0,C 180,E1 -21964.411,E2 -21964.411} C_VEL
LIN {X 0,Y 198.515,Z 437.965,A -85,B 0,C 180,E1 -21966.097,E2 -21966.097} C_VEL
LIN {X 0,Y 195.49,Z 435.479,A -85,B 0,C 180,E1 -21969.441,E2 -21969.441} C_VEL
LIN {X 0,Y 193.965,Z 432.544,A -85,B 0,C 180,E1 -21972.147,E2 -21972.147} C_VEL
LIN {X 0,Y 193.895,Z 432.607,A -85,B 0,C 180,E1 -21976.856,E2 -21976.856} C_VEL
LIN {X 0,Y 193.852,Z 433.038,A -85,B 0,C 180,E1 -21981.257,E2 -21981.257} C_VEL
LIN {X 0,Y 193.959,Z 433.835,A -85,B 0,C 180,E1 -21985.774,E2 -21985.774} C_VEL
LIN {X 0,Y 194.141,Z 435.064,A -85,B 0,C 180,E1 -21990.452,E2 -21990.452} C_VEL
LIN {X 0,Y 194.264,Z 435.581,A -85,B 0,C 180,E1 -21991.336,E2 -21991.336} C_VEL
LIN {X 0,Y 195.683,Z 438.981,A -85,B 0,C 180,E1 -21993.747,E2 -21993.747} C_VEL
LIN {X 0,Y 198.648,Z 442.416,A -85,B 0,C 180,E1 -21996.974,E2 -21996.974} C_VEL
LIN {X 0,Y 199.078,Z 443.069,A -85,B 0,C 180,E1 -21997.424,E2 -21997.424} C_VEL
LIN {X 0,Y 200.755,Z 446.814,A -85,B 0,C 180,E1 -21999.292,E2 -21999.292} C_VEL
LIN {X 0,Y 202.835,Z 449.596,A -85,B 0,C 180,E1 -22001.068,E2 -22001.068} C_VEL
LIN {X 0,Y 204.562,Z 453.408,A -85,B 0,C 180,E1 -22002.73,E2 -22002.73} C_VEL
LIN {X 0,Y 205.875,Z 455.614,A -85,B 0,C 180,E1 -22003.783,E2 -22003.783} C_VEL
LIN {X 0,Y 208.567,Z 461.883,A -85,B 0,C 180,E1 -22006.219,E2 -22006.219} C_VEL
LIN {X 0,Y 210.583,Z 467.419,A -85,B 0,C 180,E1 -22008.128,E2 -22008.128} C_VEL
LIN {X 0,Y 211.974,Z 474.146,A -85,B 0,C 180,E1 -22010.087,E2 -22010.087} C_VEL
LIN {X 0,Y 212.751,Z 483.204,A -85,B 0,C 180,E1 -22012.45,E2 -22012.45} C_VEL
LIN {X 0,Y 212.652,Z 492.818,A -85,B 0,C 180,E1 -22014.968,E2 -22014.968} C_VEL
LIN {X 0,Y 211.627,Z 501.162,A -85,B 0,C 180,E1 -22017.175,E2 -22017.175} C_VEL
LIN {X 0,Y 209.837,Z 508.654,A -85,B 0,C 180,E1 -22019.286,E2 -22019.286} C_VEL
LIN {X 0,Y 205.401,Z 517.78,A -85,B 0,C 180,E1 -22021.936,E2 -22021.936} C_VEL
LIN {X 0,Y 201.55,Z 525.208,A -85,B 0,C 180,E1 -22024.714,E2 -22024.714} C_VEL
LIN {X 0,Y 197.943,Z 532.167,A -85,B 0,C 180,E1 -22028.112,E2 -22028.112} C_VEL
LIN {X 0,Y 195.316,Z 536.858,A -85,B 0,C 180,E1 -22031.105,E2 -22031.105} C_VEL
LIN {X 0,Y 193.117,Z 540.504,A -85,B 0,C 180,E1 -22034.161,E2 -22034.161} C_VEL
LIN {X 0,Y 191.285,Z 543.907,A -85,B 0,C 180,E1 -22038.429,E2 -22038.429} C_VEL
LIN {X 0,Y 190.148,Z 544.88,A -85,B 0,C 180,E1 -22040.147,E2 -22040.147} C_VEL
LIN {X 0,Y 186.76,Z 545.744,A -85,B 0,C 180,E1 -22042.97,E2 -22042.97} C_VEL
LIN {X 0,Y 184.177,Z 545.814,A -85,B 0,C 180,E1 -22045.302,E2 -22045.302} C_VEL
LIN {X 0,Y 183.194,Z 545.585,A -85,B 0,C 180,E1 -22047.129,E2 -22047.129} C_VEL
LIN {X 0,Y 183.168,Z 545.464,A -85,B 0,C 180,E1 -22047.748,E2 -22047.748} C_VEL
LIN {X 0,Y 183.362,Z 544.734,A -85,B 0,C 180,E1 -22050.001,E2 -22050.001} C_VEL
LIN {X 0,Y 183.184,Z 542.258,A -85,B 0,C 180,E1 -22054.039,E2 -22054.039} C_VEL
LIN {X 0,Y 183.428,Z 538.729,A -85,B 0,C 180,E1 -22057.707,E2 -22057.707} C_VEL
LIN {X 0,Y 183.989,Z 534.383,A -85,B 0,C 180,E1 -22061.011,E2 -22061.011} C_VEL
LIN {X 0,Y 184.934,Z 528.809,A -85,B 0,C 180,E1 -22064.302,E2 -22064.302} C_VEL
LIN {X 0,Y 186.592,Z 521.86,A -85,B 0,C 180,E1 -22067.538,E2 -22067.538} C_VEL
LIN {X 0,Y 188.547,Z 513.212,A -85,B 0,C 180,E1 -22070.704,E2 -22070.704} C_VEL
LIN {X 0,Y 190.986,Z 503.34,A -85,B 0,C 180,E1 -22073.562,E2 -22073.562} C_VEL
LIN {X 0,Y 192.563,Z 495.575,A -85,B 0,C 180,E1 -22075.395,E2 -22075.395} C_VEL
LIN {X 0,Y 192.261,Z 484.401,A -85,B 0,C 180,E1 -22077.78,E2 -22077.78} C_VEL
LIN {X 0,Y 191.393,Z 472.584,A -85,B 0,C 180,E1 -22079.869,E2 -22079.869} C_VEL
LIN {X 0,Y 189.968,Z 460.187,A -85,B 0,C 180,E1 -22081.69,E2 -22081.69} C_VEL
LIN {X 0,Y 187.766,Z 446.791,A -85,B 0,C 180,E1 -22083.297,E2 -22083.297} C_VEL
LIN {X 0,Y 186.498,Z 440.152,A -85,B 0,C 180,E1 -22083.998,E2 -22083.998} C_VEL
LIN {X 0,Y 187.069,Z 437.574,A -85,B 0,C 180,E1 -22086.95,E2 -22086.95} C_VEL
LIN {X 0,Y 187.045,Z 435.266,A -85,B 0,C 180,E1 -22089.7,E2 -22089.7} C_VEL
LIN {X 0,Y 186.372,Z 431.688,A -85,B 0,C 180,E1 -22094.235,E2 -22094.235} C_VEL
LIN {X 0,Y 185.736,Z 427.975,A -85,B 0,C 180,E1 -22099.181,E2 -22099.181} C_VEL
LIN {X 0,Y 185.578,Z 427.376,A -85,B 0,C 180,E1 -22100.277,E2 -22100.277} C_VEL
LIN {X 0,Y 185.502,Z 427.374,A -85,B 0,C 180,E1 -22105.368,E2 -22105.368} C_VEL
LIN {X 0,Y 185.584,Z 427.366,A -85,B 0,C 180,E1 -22110.576,E2 -22110.576} C_VEL
LIN {X 0,Y 185.59,Z 427.363,A -85,B 0,C 180,E1 -22115.383,E2 -22115.383} C_VEL
LIN {X 0,Y 185.677,Z 427.353,A -85,B 0,C 180,E1 -22121.133,E2 -22121.133} C_VEL
LIN {X 0,Y 185.727,Z 427.35,A -85,B 0,C 180,E1 -22124.64,E2 -22124.64} C_VEL
LIN {X 0,Y 185.926,Z 427.322,A -85,B 0,C 180,E1 -22129.359,E2 -22129.359} C_VEL
LIN {X 0,Y 185.963,Z 427.318,A -85,B 0,C 180,E1 -22133.49,E2 -22133.49} C_VEL
LIN {X 0,Y 186.209,Z 427.284,A -85,B 0,C 180,E1 -22137.837,E2 -22137.837} C_VEL
LIN {X 0,Y 186.407,Z 427.262,A -85,B 0,C 180,E1 -22140,E2 -22140} C_VEL
LIN {X 0,Y 185.926,Z 427.318,A -85,B 0,C 180,E1 -22144.336,E2 -22144.336} C_VEL
LIN {X 0,Y 186.011,Z 427.313,A -85,B 0,C 180,E1 -22148.692,E2 -22148.692} C_VEL
LIN {X 0,Y 185.766,Z 427.336,A -85,B 0,C 180,E1 -22153.12,E2 -22153.12} C_VEL
LIN {X 0,Y 185.677,Z 427.329,A -85,B 0,C 180,E1 -22158.867,E2 -22158.867} C_VEL
LIN {X 0,Y 185.603,Z 427.363,A -85,B 0,C 180,E1 -22164.662,E2 -22164.662} C_VEL
LIN {X 0,Y 185.581,Z 427.365,A -85,B 0,C 180,E1 -22169.493,E2 -22169.493} C_VEL
LIN {X 0,Y 185.501,Z 427.355,A -85,B 0,C 180,E1 -22174.632,E2 -22174.632} C_VEL
LIN {X 0,Y 185.507,Z 427.359,A -85,B 0,C 180,E1 -22177.313,E2 -22177.313} C_VEL
LIN {X 0,Y 185.472,Z 427.377,A -85,B 0,C 180,E1 -22180.724,E2 -22180.724} C_VEL
LIN {X 0,Y 185.46,Z 427.381,A -85,B 0,C 180,E1 -22186.055,E2 -22186.055} C_VEL
LIN {X 0,Y 185.49,Z 427.365,A -85,B 0,C 180,E1 -22189.9,E2 -22189.9} C_VEL
LIN {X 0,Y 185.546,Z 427.36,A -85,B 0,C 180,E1 -22192.696,E2 -22192.696} C_VEL
LIN {X 0,Y 185.547,Z 427.372,A -85,B 0,C 180,E1 -22197.975,E2 -22197.975} C_VEL
LIN {X 0,Y 185.584,Z 427.363,A -85,B 0,C 180,E1 -22200.575,E2 -22200.575} C_VEL
LIN {X 0,Y 185.59,Z 427.363,A -85,B 0,C 180,E1 -22205.382,E2 -22205.382} C_VEL
LIN {X 0,Y 185.609,Z 427.363,A -85,B 0,C 180,E1 -22210.075,E2 -22210.075} C_VEL
LIN {X 0,Y 185.727,Z 427.353,A -85,B 0,C 180,E1 -22214.639,E2 -22214.639} C_VEL
LIN {X 0,Y 185.944,Z 427.319,A -85,B 0,C 180,E1 -22219.328,E2 -22219.328} C_VEL
LIN {X 0,Y 185.971,Z 427.317,A -85,B 0,C 180,E1 -22223.489,E2 -22223.489} C_VEL
LIN {X 0,Y 186.209,Z 427.285,A -85,B 0,C 180,E1 -22227.836,E2 -22227.836} C_VEL
LIN {X 0,Y 186.407,Z 427.268,A -85,B 0,C 180,E1 -22229.999,E2 -22229.999} C_VEL
LIN {X 0,Y 185.852,Z 427.333,A -85,B 0,C 180,E1 -22234.337,E2 -22234.337} C_VEL
LIN {X 0,Y 185.766,Z 427.347,A -85,B 0,C 180,E1 -22236.516,E2 -22236.516} C_VEL
LIN {X 0,Y 185.442,Z 427.508,A -85,B 0,C 180,E1 -22239.015,E2 -22239.015} C_VEL
LIN {X 0,Y 188.794,Z 439.869,A -85,B 0,C 180,E1 -22240.513,E2 -22240.513} C_VEL
LIN {X 0,Y 191.443,Z 451.279,A -85,B 0,C 180,E1 -22242.185,E2 -22242.185} C_VEL
LIN {X 0,Y 193.564,Z 463.044,A -85,B 0,C 180,E1 -22244.189,E2 -22244.189} C_VEL
LIN {X 0,Y 195.019,Z 474.601,A -85,B 0,C 180,E1 -22246.486,E2 -22246.486} C_VEL
LIN {X 0,Y 192.63,Z 485.798,A -85,B 0,C 180,E1 -22248.849,E2 -22248.849} C_VEL
LIN {X 0,Y 190.384,Z 495.355,A -85,B 0,C 180,E1 -22251.378,E2 -22251.378} C_VEL
LIN {X 0,Y 188.273,Z 504.05,A -85,B 0,C 180,E1 -22254.242,E2 -22254.242} C_VEL
LIN {X 0,Y 186.409,Z 511.816,A -85,B 0,C 180,E1 -22257.478,E2 -22257.478} C_VEL
LIN {X 0,Y 184.934,Z 518.242,A -85,B 0,C 180,E1 -22260.865,E2 -22260.865} C_VEL
LIN {X 0,Y 183.992,Z 522.782,A -85,B 0,C 180,E1 -22263.9,E2 -22263.9} C_VEL
LIN {X 0,Y 183.16,Z 527.281,A -85,B 0,C 180,E1 -22267.873,E2 -22267.873} C_VEL
LIN {X 0,Y 182.808,Z 529.614,A -85,B 0,C 180,E1 -22270.809,E2 -22270.809} C_VEL
LIN {X 0,Y 182.752,Z 531.251,A -85,B 0,C 180,E1 -22273.804,E2 -22273.804} C_VEL
LIN {X 0,Y 183.009,Z 532.179,A -85,B 0,C 180,E1 -22276.855,E2 -22276.855} C_VEL
LIN {X 0,Y 183.657,Z 532.318,A -85,B 0,C 180,E1 -22279.935,E2 -22279.935} C_VEL
LIN {X 0,Y 184.68,Z 531.691,A -85,B 0,C 180,E1 -22283.048,E2 -22283.048} C_VEL
LIN {X 0,Y 186.127,Z 530.262,A -85,B 0,C 180,E1 -22286.169,E2 -22286.169} C_VEL
LIN {X 0,Y 188.027,Z 527.974,A -85,B 0,C 180,E1 -22289.279,E2 -22289.279} C_VEL
LIN {X 0,Y 191.053,Z 523.724,A -85,B 0,C 180,E1 -22293.143,E2 -22293.143} C_VEL
LIN {X 0,Y 194.561,Z 518.43,A -85,B 0,C 180,E1 -22296.588,E2 -22296.588} C_VEL
LIN {X 0,Y 198.617,Z 511.922,A -85,B 0,C 180,E1 -22299.73,E2 -22299.73} C_VEL
LIN {X 0,Y 202.404,Z 505.128,A -85,B 0,C 180,E1 -22302.287,E2 -22302.287} C_VEL
LIN {X 0,Y 207.015,Z 495.9,A -85,B 0,C 180,E1 -22304.998,E2 -22304.998} C_VEL
LIN {X 0,Y 208.648,Z 492.366,A -85,B 0,C 180,E1 -22305.865,E2 -22305.865} C_VEL
LIN {X 0,Y 209.116,Z 490.551,A -85,B 0,C 180,E1 -22306.393,E2 -22306.393} C_VEL
LIN {X 0,Y 209.356,Z 482.79,A -85,B 0,C 180,E1 -22308.919,E2 -22308.919} C_VEL
LIN {X 0,Y 208.489,Z 474.252,A -85,B 0,C 180,E1 -22311.763,E2 -22311.763} C_VEL
LIN {X 0,Y 207.216,Z 467.395,A -85,B 0,C 180,E1 -22314.16,E2 -22314.16} C_VEL
LIN {X 0,Y 205.055,Z 461.324,A -85,B 0,C 180,E1 -22316.652,E2 -22316.652} C_VEL
LIN {X 0,Y 202.723,Z 456.294,A -85,B 0,C 180,E1 -22319.067,E2 -22319.067} C_VEL
LIN {X 0,Y 200.03,Z 450.689,A -85,B 0,C 180,E1 -22322.014,E2 -22322.014} C_VEL
LIN {X 0,Y 199.037,Z 449.212,A -85,B 0,C 180,E1 -22323.037,E2 -22323.037} C_VEL
LIN {X 0,Y 197.046,Z 446.84,A -85,B 0,C 180,E1 -22325.052,E2 -22325.052} C_VEL
LIN {X 0,Y 196.279,Z 445.074,A -85,B 0,C 180,E1 -22326.167,E2 -22326.167} C_VEL
LIN {X 0,Y 192.624,Z 440.795,A -85,B 0,C 180,E1 -22331.199,E2 -22331.199} C_VEL
LIN {X 0,Y 191.941,Z 439.36,A -85,B 0,C 180,E1 -22332.691,E2 -22332.691} C_VEL
LIN {X 0,Y 190.017,Z 438.573,A -85,B 0,C 180,E1 -22337.211,E2 -22337.211} C_VEL
LIN {X 0,Y 189.466,Z 438.737,A -85,B 0,C 180,E1 -22341.979,E2 -22341.979} C_VEL
LIN {X 0,Y 190.293,Z 440.104,A -85,B 0,C 180,E1 -22346.604,E2 -22346.604} C_VEL
LIN {X 0,Y 192.262,Z 442.206,A -85,B 0,C 180,E1 -22350.781,E2 -22350.781} C_VEL
LIN {X 0,Y 193.904,Z 446.328,A -85,B 0,C 180,E1 -22353.946,E2 -22353.946} C_VEL
LIN {X 0,Y 195.928,Z 448.684,A -85,B 0,C 180,E1 -22356.29,E2 -22356.29} C_VEL
LIN {X 0,Y 198.638,Z 454.208,A -85,B 0,C 180,E1 -22359.558,E2 -22359.558} C_VEL
LIN {X 0,Y 199.454,Z 455.255,A -85,B 0,C 180,E1 -22360.304,E2 -22360.304} C_VEL
LIN {X 0,Y 201.331,Z 459.672,A -85,B 0,C 180,E1 -22362.403,E2 -22362.403} C_VEL
LIN {X 0,Y 203.927,Z 465.721,A -85,B 0,C 180,E1 -22365.057,E2 -22365.057} C_VEL
LIN {X 0,Y 206.221,Z 473.355,A -85,B 0,C 180,E1 -22367.837,E2 -22367.837} C_VEL
LIN {X 0,Y 207.101,Z 480.884,A -85,B 0,C 180,E1 -22370.074,E2 -22370.074} C_VEL
LIN {X 0,Y 207.121,Z 491.309,A -85,B 0,C 180,E1 -22372.971,E2 -22372.971} C_VEL
LIN {X 0,Y 206.135,Z 500.152,A -85,B 0,C 180,E1 -22375.477,E2 -22375.477} C_VEL
LIN {X 0,Y 204.381,Z 507.983,A -85,B 0,C 180,E1 -22377.793,E2 -22377.793} C_VEL
LIN {X 0,Y 201.53,Z 514.276,A -85,B 0,C 180,E1 -22379.626,E2 -22379.626} C_VEL
LIN {X 0,Y 197.828,Z 521.077,A -85,B 0,C 180,E1 -22381.92,E2 -22381.92} C_VEL
LIN {X 0,Y 194.572,Z 526.816,A -85,B 0,C 180,E1 -22384.315,E2 -22384.315} C_VEL
LIN {X 0,Y 191.355,Z 532.479,A -85,B 0,C 180,E1 -22387.318,E2 -22387.318} C_VEL
LIN {X 0,Y 188.62,Z 537.047,A -85,B 0,C 180,E1 -22390.408,E2 -22390.408} C_VEL
LIN {X 0,Y 185.652,Z 541.526,A -85,B 0,C 180,E1 -22394.635,E2 -22394.635} C_VEL
LIN {X 0,Y 184.028,Z 544.407,A -85,B 0,C 180,E1 -22398.993,E2 -22398.993} C_VEL
LIN {X 0,Y 183.21,Z 545.683,A -85,B 0,C 180,E1 -22403.393,E2 -22403.393} C_VEL
LIN {X 0,Y 183.168,Z 545.464,A -85,B 0,C 180,E1 -22407.748,E2 -22407.748} C_VEL
LIN {X 0,Y 182.944,Z 545.145,A -85,B 0,C 180,E1 -22408.971,E2 -22408.971} C_VEL
LIN {X 0,Y 182.169,Z 544.646,A -85,B 0,C 180,E1 -22410.173,E2 -22410.173} C_VEL
LIN {X 0,Y 179.737,Z 543.202,A -85,B 0,C 180,E1 -22412.529,E2 -22412.529} C_VEL
LIN {X 0,Y 177.276,Z 541.215,A -85,B 0,C 180,E1 -22414.918,E2 -22414.918} C_VEL
LIN {X 0,Y 176.313,Z 539.432,A -85,B 0,C 180,E1 -22416.754,E2 -22416.754} C_VEL
LIN {X 0,Y 176.288,Z 538.763,A -85,B 0,C 180,E1 -22417.371,E2 -22417.371} C_VEL
LIN {X 0,Y 176.981,Z 533.602,A -85,B 0,C 180,E1 -22421.453,E2 -22421.453} C_VEL
LIN {X 0,Y 178.293,Z 526.789,A -85,B 0,C 180,E1 -22425.432,E2 -22425.432} C_VEL
LIN {X 0,Y 180.061,Z 519.379,A -85,B 0,C 180,E1 -22428.785,E2 -22428.785} C_VEL
LIN {X 0,Y 181.724,Z 512.32,A -85,B 0,C 180,E1 -22431.371,E2 -22431.371} C_VEL
LIN {X 0,Y 184.176,Z 502.92,A -85,B 0,C 180,E1 -22434.159,E2 -22434.159} C_VEL
LIN {X 0,Y 185.612,Z 496.177,A -85,B 0,C 180,E1 -22435.814,E2 -22435.814} C_VEL
LIN {X 0,Y 185.389,Z 484.636,A -85,B 0,C 180,E1 -22438.404,E2 -22438.404} C_VEL
LIN {X 0,Y 184.646,Z 473.693,A -85,B 0,C 180,E1 -22440.458,E2 -22440.458} C_VEL
LIN {X 0,Y 183.27,Z 460.725,A -85,B 0,C 180,E1 -22442.472,E2 -22442.472} C_VEL
LIN {X 0,Y 181.099,Z 447.379,A -85,B 0,C 180,E1 -22444.169,E2 -22444.169} C_VEL
LIN {X 0,Y 179.648,Z 439.925,A -85,B 0,C 180,E1 -22444.954,E2 -22444.954} C_VEL
LIN {X 0,Y 180.02,Z 438.022,A -85,B 0,C 180,E1 -22447.238,E2 -22447.238} C_VEL
LIN {X 0,Y 179.922,Z 435.717,A -85,B 0,C 180,E1 -22450.128,E2 -22450.128} C_VEL
LIN {X 0,Y 179.194,Z 431.952,A -85,B 0,C 180,E1 -22455.092,E2 -22455.092} C_VEL
LIN {X 0,Y 178.535,Z 428.254,A -85,B 0,C 180,E1 -22460.415,E2 -22460.415} C_VEL
LIN {X 0,Y 178.489,Z 428.251,A -85,B 0,C 180,E1 -22466.547,E2 -22466.547} C_VEL
LIN {X 0,Y 178.525,Z 428.245,A -85,B 0,C 180,E1 -22470.006,E2 -22470.006} C_VEL
LIN {X 0,Y 178.537,Z 428.238,A -85,B 0,C 180,E1 -22474.876,E2 -22474.876} C_VEL
LIN {X 0,Y 178.626,Z 428.232,A -85,B 0,C 180,E1 -22480.784,E2 -22480.784} C_VEL
LIN {X 0,Y 178.668,Z 428.228,A -85,B 0,C 180,E1 -22484.017,E2 -22484.017} C_VEL
LIN {X 0,Y 178.864,Z 428.2,A -85,B 0,C 180,E1 -22489.21,E2 -22489.21} C_VEL
LIN {X 0,Y 178.927,Z 428.196,A -85,B 0,C 180,E1 -22493.233,E2 -22493.233} C_VEL
LIN {X 0,Y 179.155,Z 428.163,A -85,B 0,C 180,E1 -22497.752,E2 -22497.752} C_VEL
LIN {X 0,Y 179.37,Z 428.139,A -85,B 0,C 180,E1 -22500,E2 -22500} C_VEL
LIN {X 0,Y 178.874,Z 428.196,A -85,B 0,C 180,E1 -22504.507,E2 -22504.507} C_VEL
LIN {X 0,Y 178.962,Z 428.192,A -85,B 0,C 180,E1 -22509.038,E2 -22509.038} C_VEL
LIN {X 0,Y 178.683,Z 428.216,A -85,B 0,C 180,E1 -22513.65,E2 -22513.65} C_VEL
LIN {X 0,Y 178.625,Z 428.208,A -85,B 0,C 180,E1 -22519.216,E2 -22519.216} C_VEL
LIN {X 0,Y 178.537,Z 428.245,A -85,B 0,C 180,E1 -22525.124,E2 -22525.124} C_VEL
LIN {X 0,Y 178.481,Z 428.246,A -85,B 0,C 180,E1 -22530.79,E2 -22530.79} C_VEL
LIN {X 0,Y 178.487,Z 428.231,A -85,B 0,C 180,E1 -22534.219,E2 -22534.219} C_VEL
LIN {X 0,Y 178.396,Z 428.252,A -85,B 0,C 180,E1 -22539.074,E2 -22539.074} C_VEL
LIN {X 0,Y 178.399,Z 428.259,A -85,B 0,C 180,E1 -22542.045,E2 -22542.045} C_VEL
LIN {X 0,Y 178.395,Z 428.261,A -85,B 0,C 180,E1 -22545.164,E2 -22545.164} C_VEL
LIN {X 0,Y 178.411,Z 428.251,A -85,B 0,C 180,E1 -22548.456,E2 -22548.456} C_VEL
LIN {X 0,Y 178.465,Z 428.237,A -85,B 0,C 180,E1 -22551.962,E2 -22551.962} C_VEL
LIN {X 0,Y 178.493,Z 428.251,A -85,B 0,C 180,E1 -22556.547,E2 -22556.547} C_VEL
LIN {X 0,Y 178.525,Z 428.245,A -85,B 0,C 180,E1 -22560.006,E2 -22560.006} C_VEL
LIN {X 0,Y 178.536,Z 428.241,A -85,B 0,C 180,E1 -22564.875,E2 -22564.875} C_VEL
LIN {X 0,Y 178.625,Z 428.228,A -85,B 0,C 180,E1 -22570.783,E2 -22570.783} C_VEL
LIN {X 0,Y 178.668,Z 428.228,A -85,B 0,C 180,E1 -22574.016,E2 -22574.016} C_VEL
LIN {X 0,Y 178.897,Z 428.197,A -85,B 0,C 180,E1 -22579.153,E2 -22579.153} C_VEL
LIN {X 0,Y 178.936,Z 428.193,A -85,B 0,C 180,E1 -22583.232,E2 -22583.232} C_VEL
LIN {X 0,Y 179.155,Z 428.163,A -85,B 0,C 180,E1 -22587.751,E2 -22587.751} C_VEL
LIN {X 0,Y 179.369,Z 428.145,A -85,B 0,C 180,E1 -22589.999,E2 -22589.999} C_VEL
LIN {X 0,Y 178.788,Z 428.214,A -85,B 0,C 180,E1 -22594.508,E2 -22594.508} C_VEL
LIN {X 0,Y 178.519,Z 428.244,A -85,B 0,C 180,E1 -22597.99,E2 -22597.99} C_VEL
LIN {X 0,Y 182.401,Z 442.151,A -85,B 0,C 180,E1 -22599.875,E2 -22599.875} C_VEL
LIN {X 0,Y 184.852,Z 452.965,A -85,B 0,C 180,E1 -22601.556,E2 -22601.556} C_VEL
LIN {X 0,Y 186.812,Z 464.295,A -85,B 0,C 180,E1 -22603.598,E2 -22603.598} C_VEL
LIN {X 0,Y 188.149,Z 475.671,A -85,B 0,C 180,E1 -22605.99,E2 -22605.99} C_VEL
LIN {X 0,Y 185.626,Z 486.775,A -85,B 0,C 180,E1 -22608.442,E2 -22608.442} C_VEL
LIN {X 0,Y 183.358,Z 496.199,A -85,B 0,C 180,E1 -22611.058,E2 -22611.058} C_VEL
LIN {X 0,Y 181.183,Z 504.777,A -85,B 0,C 180,E1 -22614.034,E2 -22614.034} C_VEL
LIN {X 0,Y 179.171,Z 512.825,A -85,B 0,C 180,E1 -22617.572,E2 -22617.572} C_VEL
LIN {X 0,Y 177.789,Z 518.833,A -85,B 0,C 180,E1 -22620.922,E2 -22620.922} C_VEL
LIN {X 0,Y 176.916,Z 522.935,A -85,B 0,C 180,E1 -22623.789,E2 -22623.789} C_VEL
LIN {X 0,Y 176.199,Z 526.656,A -85,B 0,C 180,E1 -22627.086,E2 -22627.086} C_VEL
LIN {X 0,Y 175.725,Z 529.533,A -85,B 0,C 180,E1 -22630.545,E2 -22630.545} C_VEL
LIN {X 0,Y 175.655,Z 531.427,A -85,B 0,C 180,E1 -22633.93,E2 -22633.93} C_VEL
LIN {X 0,Y 175.976,Z 532.439,A -85,B 0,C 180,E1 -22637.24,E2 -22637.24} C_VEL
LIN {X 0,Y 176.693,Z 532.615,A -85,B 0,C 180,E1 -22640.476,E2 -22640.476} C_VEL
LIN {X 0,Y 177.788,Z 532.047,A -85,B 0,C 180,E1 -22643.633,E2 -22643.633} C_VEL
LIN {X 0,Y 179.243,Z 530.775,A -85,B 0,C 180,E1 -22646.706,E2 -22646.706} C_VEL
LIN {X 0,Y 182.043,Z 527.626,A -85,B 0,C 180,E1 -22651.002,E2 -22651.002} C_VEL
LIN {X 0,Y 185.759,Z 522.798,A -85,B 0,C 180,E1 -22655.23,E2 -22655.23} C_VEL
LIN {X 0,Y 189.15,Z 517.957,A -85,B 0,C 180,E1 -22658.26,E2 -22658.26} C_VEL
LIN {X 0,Y 193.902,Z 510.562,A -85,B 0,C 180,E1 -22661.718,E2 -22661.718} C_VEL
LIN {X 0,Y 198.225,Z 503.089,A -85,B 0,C 180,E1 -22664.416,E2 -22664.416} C_VEL
LIN {X 0,Y 202.257,Z 495.34,A -85,B 0,C 180,E1 -22666.635,E2 -22666.635} C_VEL
LIN {X 0,Y 203.115,Z 493.41,A -85,B 0,C 180,E1 -22667.138,E2 -22667.138} C_VEL
LIN {X 0,Y 203.696,Z 486.436,A -85,B 0,C 180,E1 -22669.564,E2 -22669.564} C_VEL
LIN {X 0,Y 203.307,Z 478.449,A -85,B 0,C 180,E1 -22672.427,E2 -22672.427} C_VEL
LIN {X 0,Y 202.265,Z 471.537,A -85,B 0,C 180,E1 -22675.017,E2 -22675.017} C_VEL
LIN {X 0,Y 200.789,Z 466.692,A -85,B 0,C 180,E1 -22677.174,E2 -22677.174} C_VEL
LIN {X 0,Y 197.668,Z 459.097,A -85,B 0,C 180,E1 -22681.148,E2 -22681.148} C_VEL
LIN {X 0,Y 196.139,Z 455.895,A -85,B 0,C 180,E1 -22683.082,E2 -22683.082} C_VEL
LIN {X 0,Y 194.413,Z 453.659,A -85,B 0,C 180,E1 -22685.065,E2 -22685.065} C_VEL
LIN {X 0,Y 193.644,Z 451.975,A -85,B 0,C 180,E1 -22686.251,E2 -22686.251} C_VEL
LIN {X 0,Y 190.148,Z 447.062,A -85,B 0,C 180,E1 -22691.933,E2 -22691.933} C_VEL
LIN {X 0,Y 189.873,Z 446.141,A -85,B 0,C 180,E1 -22692.832,E2 -22692.832} C_VEL
LIN {X 0,Y 188.107,Z 445.402,A -85,B 0,C 180,E1 -22697.391,E2 -22697.391} C_VEL
LIN {X 0,Y 187.622,Z 445.603,A -85,B 0,C 180,E1 -22701.999,E2 -22701.999} C_VEL
LIN {X 0,Y 188.396,Z 446.975,A -85,B 0,C 180,E1 -22706.593,E2 -22706.593} C_VEL
LIN {X 0,Y 189.962,Z 448.942,A -85,B 0,C 180,E1 -22710.388,E2 -22710.388} C_VEL
LIN {X 0,Y 191.304,Z 452.705,A -85,B 0,C 180,E1 -22713.44,E2 -22713.44} C_VEL
LIN {X 0,Y 192.95,Z 454.855,A -85,B 0,C 180,E1 -22715.647,E2 -22715.647} C_VEL
LIN {X 0,Y 196.226,Z 462.1,A -85,B 0,C 180,E1 -22720.142,E2 -22720.142} C_VEL
LIN {X 0,Y 198.04,Z 466.434,A -85,B 0,C 180,E1 -22722.398,E2 -22722.398} C_VEL
LIN {X 0,Y 200.653,Z 474.546,A -85,B 0,C 180,E1 -22725.891,E2 -22725.891} C_VEL
LIN {X 0,Y 201.514,Z 479.239,A -85,B 0,C 180,E1 -22727.568,E2 -22727.568} C_VEL
LIN {X 0,Y 201.802,Z 486.112,A -85,B 0,C 180,E1 -22729.686,E2 -22729.686} C_VEL
LIN {X 0,Y 201.311,Z 494.929,A -85,B 0,C 180,E1 -22732.344,E2 -22732.344} C_VEL
LIN {X 0,Y 200.123,Z 502.613,A -85,B 0,C 180,E1 -22734.681,E2 -22734.681} C_VEL
LIN {X 0,Y 197.848,Z 510.586,A -85,B 0,C 180,E1 -22737.201,E2 -22737.201} C_VEL
LIN {X 0,Y 193.083,Z 519.206,A -85,B 0,C 180,E1 -22739.969,E2 -22739.969} C_VEL
LIN {X 0,Y 188.856,Z 526.269,A -85,B 0,C 180,E1 -22742.88,E2 -22742.88} C_VEL
LIN {X 0,Y 184.817,Z 532.802,A -85,B 0,C 180,E1 -22746.468,E2 -22746.468} C_VEL
LIN {X 0,Y 181.94,Z 537.213,A -85,B 0,C 180,E1 -22749.657,E2 -22749.657} C_VEL
LIN {X 0,Y 178.785,Z 541.55,A -85,B 0,C 180,E1 -22754.029,E2 -22754.029} C_VEL
LIN {X 0,Y 177.79,Z 543.122,A -85,B 0,C 180,E1 -22756.281,E2 -22756.281} C_VEL
LIN {X 0,Y 176.466,Z 545.035,A -85,B 0,C 180,E1 -22760.834,E2 -22760.834} C_VEL
LIN {X 0,Y 176.007,Z 545.453,A -85,B 0,C 180,E1 -22765.42,E2 -22765.42} C_VEL
LIN {X 0,Y 176.098,Z 545.066,A -85,B 0,C 180,E1 -22767.747,E2 -22767.747} C_VEL
LIN {X 0,Y 176.278,Z 544.283,A -85,B 0,C 180,E1 -22770.001,E2 -22770.001} C_VEL
LIN {X 0,Y 176.111,Z 541.928,A -85,B 0,C 180,E1 -22773.911,E2 -22773.911} C_VEL
LIN {X 0,Y 176.288,Z 538.763,A -85,B 0,C 180,E1 -22777.371,E2 -22777.371} C_VEL
LIN {X 0,Y 175.859,Z 536.689,A -85,B 0,C 180,E1 -22779.158,E2 -22779.158} C_VEL
LIN {X 0,Y 173.576,Z 532.681,A -85,B 0,C 180,E1 -22782.033,E2 -22782.033} C_VEL
LIN {X 0,Y 171.601,Z 528.011,A -85,B 0,C 180,E1 -22784.879,E2 -22784.879} C_VEL
LIN {X 0,Y 171.679,Z 524.837,A -85,B 0,C 180,E1 -22786.569,E2 -22786.569} C_VEL
LIN {X 0,Y 173.681,Z 516.801,A -85,B 0,C 180,E1 -22790.119,E2 -22790.119} C_VEL
LIN {X 0,Y 175.764,Z 508.492,A -85,B 0,C 180,E1 -22793.041,E2 -22793.041} C_VEL
LIN {X 0,Y 178.172,Z 499.008,A -85,B 0,C 180,E1 -22795.716,E2 -22795.716} C_VEL
LIN {X 0,Y 178.666,Z 495.548,A -85,B 0,C 180,E1 -22796.581,E2 -22796.581} C_VEL
LIN {X 0,Y 178.538,Z 484.958,A -85,B 0,C 180,E1 -22799.049,E2 -22799.049} C_VEL
LIN {X 0,Y 177.77,Z 473.133,A -85,B 0,C 180,E1 -22801.358,E2 -22801.358} C_VEL
LIN {X 0,Y 176.334,Z 460.053,A -85,B 0,C 180,E1 -22803.464,E2 -22803.464} C_VEL
LIN {X 0,Y 174.305,Z 447.29,A -85,B 0,C 180,E1 -22805.163,E2 -22805.163} C_VEL
LIN {X 0,Y 172.84,Z 439.63,A -85,B 0,C 180,E1 -22806.087,E2 -22806.087} C_VEL
LIN {X 0,Y 172.914,Z 436.996,A -85,B 0,C 180,E1 -22809.443,E2 -22809.443} C_VEL
LIN {X 0,Y 172.328,Z 433.727,A -85,B 0,C 180,E1 -22813.893,E2 -22813.893} C_VEL
LIN {X 0,Y 171.684,Z 430.105,A -85,B 0,C 180,E1 -22819.082,E2 -22819.082} C_VEL
LIN {X 0,Y 171.514,Z 429.128,A -85,B 0,C 180,E1 -22820.778,E2 -22820.778} C_VEL
LIN {X 0,Y 171.403,Z 429.127,A -85,B 0,C 180,E1 -22825.091,E2 -22825.091} C_VEL
LIN {X 0,Y 171.452,Z 429.126,A -85,B 0,C 180,E1 -22830.535,E2 -22830.535} C_VEL
LIN {X 0,Y 171.46,Z 429.124,A -85,B 0,C 180,E1 -22835.802,E2 -22835.802} C_VEL
LIN {X 0,Y 171.582,Z 429.109,A -85,B 0,C 180,E1 -22840.872,E2 -22840.872} C_VEL
LIN {X 0,Y 171.612,Z 429.107,A -85,B 0,C 180,E1 -22845.776,E2 -22845.776} C_VEL
LIN {X 0,Y 171.891,Z 429.07,A -85,B 0,C 180,E1 -22850.587,E2 -22850.587} C_VEL
LIN {X 0,Y 171.823,Z 429.075,A -85,B 0,C 180,E1 -22855.307,E2 -22855.307} C_VEL
LIN {X 0,Y 172.333,Z 429.015,A -85,B 0,C 180,E1 -22860,E2 -22860} C_VEL
LIN {X 0,Y 171.823,Z 429.074,A -85,B 0,C 180,E1 -22864.692,E2 -22864.692} C_VEL
LIN {X 0,Y 171.891,Z 429.071,A -85,B 0,C 180,E1 -22869.413,E2 -22869.413} C_VEL
LIN {X 0,Y 171.596,Z 429.098,A -85,B 0,C 180,E1 -22874.225,E2 -22874.225} C_VEL
LIN {X 0,Y 171.547,Z 429.091,A -85,B 0,C 180,E1 -22879.562,E2 -22879.562} C_VEL
LIN {X 0,Y 171.471,Z 429.124,A -85,B 0,C 180,E1 -22885.616,E2 -22885.616} C_VEL
LIN {X 0,Y 171.444,Z 429.124,A -85,B 0,C 180,E1 -22890.587,E2 -22890.587} C_VEL
LIN {X 0,Y 171.394,Z 429.107,A -85,B 0,C 180,E1 -22895.034,E2 -22895.034} C_VEL
LIN {X 0,Y 171.359,Z 429.126,A -85,B 0,C 180,E1 -22898.807,E2 -22898.807} C_VEL
LIN {X 0,Y 171.322,Z 429.144,A -85,B 0,C 180,E1 -22904.217,E2 -22904.217} C_VEL
LIN {X 0,Y 171.345,Z 429.127,A -85,B 0,C 180,E1 -22908.984,E2 -22908.984} C_VEL
LIN {X 0,Y 171.415,Z 429.115,A -85,B 0,C 180,E1 -22912.047,E2 -22912.047} C_VEL
LIN {X 0,Y 171.413,Z 429.131,A -85,B 0,C 180,E1 -22915.086,E2 -22915.086} C_VEL
LIN {X 0,Y 171.451,Z 429.123,A -85,B 0,C 180,E1 -22920.534,E2 -22920.534} C_VEL
LIN {X 0,Y 171.46,Z 429.124,A -85,B 0,C 180,E1 -22925.801,E2 -22925.801} C_VEL
LIN {X 0,Y 171.581,Z 429.105,A -85,B 0,C 180,E1 -22930.871,E2 -22930.871} C_VEL
LIN {X 0,Y 171.612,Z 429.11,A -85,B 0,C 180,E1 -22935.775,E2 -22935.775} C_VEL
LIN {X 0,Y 171.912,Z 429.071,A -85,B 0,C 180,E1 -22940.588,E2 -22940.588} C_VEL
LIN {X 0,Y 171.825,Z 429.069,A -85,B 0,C 180,E1 -22945.307,E2 -22945.307} C_VEL
LIN {X 0,Y 172.331,Z 429.022,A -85,B 0,C 180,E1 -22949.999,E2 -22949.999} C_VEL
LIN {X 0,Y 171.72,Z 429.096,A -85,B 0,C 180,E1 -22954.694,E2 -22954.694} C_VEL
LIN {X 0,Y 171.609,Z 429.143,A -85,B 0,C 180,E1 -22956.982,E2 -22956.982} C_VEL
LIN {X 0,Y 174.66,Z 439.037,A -85,B 0,C 180,E1 -22958.386,E2 -22958.386} C_VEL
LIN {X 0,Y 177.528,Z 450.882,A -85,B 0,C 180,E1 -22960.261,E2 -22960.261} C_VEL
LIN {X 0,Y 179.637,Z 462.709,A -85,B 0,C 180,E1 -22962.425,E2 -22962.425} C_VEL
LIN {X 0,Y 181.114,Z 474.304,A -85,B 0,C 180,E1 -22964.896,E2 -22964.896} C_VEL
LIN {X 0,Y 181.259,Z 476.728,A -85,B 0,C 180,E1 -22965.459,E2 -22965.459} C_VEL
LIN {X 0,Y 178.629,Z 487.875,A -85,B 0,C 180,E1 -22968.048,E2 -22968.048} C_VEL
LIN {X 0,Y 176.555,Z 496.046,A -85,B 0,C 180,E1 -22970.416,E2 -22970.416} C_VEL
LIN {X 0,Y 174.096,Z 505.448,A -85,B 0,C 180,E1 -22973.808,E2 -22973.808} C_VEL
LIN {X 0,Y 172.117,Z 513.136,A -85,B 0,C 180,E1 -22977.345,E2 -22977.345} C_VEL
LIN {X 0,Y 170.522,Z 519.823,A -85,B 0,C 180,E1 -22981.281,E2 -22981.281} C_VEL
LIN {X 0,Y 169.411,Z 525.177,A -85,B 0,C 180,E1 -22985.505,E2 -22985.505} C_VEL
LIN {X 0,Y 168.842,Z 528.182,A -85,B 0,C 180,E1 -22988.634,E2 -22988.634} C_VEL
LIN {X 0,Y 168.55,Z 530.45,A -85,B 0,C 180,E1 -22991.846,E2 -22991.846} C_VEL
LIN {X 0,Y 168.607,Z 531.984,A -85,B 0,C 180,E1 -22995.12,E2 -22995.12} C_VEL
LIN {X 0,Y 169.103,Z 532.804,A -85,B 0,C 180,E1 -22998.423,E2 -22998.423} C_VEL
LIN {X 0,Y 169.98,Z 532.885,A -85,B 0,C 180,E1 -23001.772,E2 -23001.772} C_VEL
LIN {X 0,Y 171.3,Z 532.15,A -85,B 0,C 180,E1 -23005.138,E2 -23005.138} C_VEL
LIN {X 0,Y 173.108,Z 530.612,A -85,B 0,C 180,E1 -23008.491,E2 -23008.491} C_VEL
LIN {X 0,Y 175.407,Z 528.215,A -85,B 0,C 180,E1 -23011.817,E2 -23011.817} C_VEL
LIN {X 0,Y 178.232,Z 524.882,A -85,B 0,C 180,E1 -23015.081,E2 -23015.081} C_VEL
LIN {X 0,Y 182.662,Z 519.18,A -85,B 0,C 180,E1 -23019.057,E2 -23019.057} C_VEL
LIN {X 0,Y 187.538,Z 512.257,A -85,B 0,C 180,E1 -23022.555,E2 -23022.555} C_VEL
LIN {X 0,Y 192.548,Z 504.169,A -85,B 0,C 180,E1 -23025.622,E2 -23025.622} C_VEL
LIN {X 0,Y 197.312,Z 495.465,A -85,B 0,C 180,E1 -23028.182,E2 -23028.182} C_VEL
LIN {X 0,Y 198.08,Z 488.439,A -85,B 0,C 180,E1 -23030.813,E2 -23030.813} C_VEL
LIN {X 0,Y 197.906,Z 480.515,A -85,B 0,C 180,E1 -23033.884,E2 -23033.884} C_VEL
LIN {X 0,Y 197.026,Z 474.287,A -85,B 0,C 180,E1 -23036.535,E2 -23036.535} C_VEL
LIN {X 0,Y 194.856,Z 467.645,A -85,B 0,C 180,E1 -23040,E2 -23040} C_VEL
LIN {X 0,Y 192.884,Z 462.53,A -85,B 0,C 180,E1 -23043.089,E2 -23043.089} C_VEL
LIN {X 0,Y 189.971,Z 457.524,A -85,B 0,C 180,E1 -23047.44,E2 -23047.44} C_VEL
LIN {X 0,Y 187.43,Z 453.012,A -85,B 0,C 180,E1 -23052.866,E2 -23052.866} C_VEL
LIN {X 0,Y 185.812,Z 452.132,A -85,B 0,C 180,E1 -23057.613,E2 -23057.613} C_VEL
LIN {X 0,Y 185.443,Z 452.375,A -85,B 0,C 180,E1 -23062.271,E2 -23062.271} C_VEL
LIN {X 0,Y 186.219,Z 453.85,A -85,B 0,C 180,E1 -23066.929,E2 -23066.929} C_VEL
LIN {X 0,Y 187.053,Z 454.936,A -85,B 0,C 180,E1 -23069.238,E2 -23069.238} C_VEL
LIN {X 0,Y 189.998,Z 461.605,A -85,B 0,C 180,E1 -23075.535,E2 -23075.535} C_VEL
LIN {X 0,Y 192.27,Z 467.293,A -85,B 0,C 180,E1 -23079.268,E2 -23079.268} C_VEL
LIN {X 0,Y 193.816,Z 471.47,A -85,B 0,C 180,E1 -23081.584,E2 -23081.584} C_VEL
LIN {X 0,Y 195.905,Z 479.079,A -85,B 0,C 180,E1 -23085.114,E2 -23085.114} C_VEL
LIN {X 0,Y 196.435,Z 482.971,A -85,B 0,C 180,E1 -23086.624,E2 -23086.624} C_VEL
LIN {X 0,Y 196.411,Z 489.251,A -85,B 0,C 180,E1 -23088.714,E2 -23088.714} C_VEL
LIN {X 0,Y 195.453,Z 498.391,A -85,B 0,C 180,E1 -23091.666,E2 -23091.666} C_VEL
LIN {X 0,Y 193.821,Z 505.955,A -85,B 0,C 180,E1 -23094.146,E2 -23094.146} C_VEL
LIN {X 0,Y 191.957,Z 511.62,A -85,B 0,C 180,E1 -23096.06,E2 -23096.06} C_VEL
LIN {X 0,Y 187.022,Z 519.981,A -85,B 0,C 180,E1 -23098.89,E2 -23098.89} C_VEL
LIN {X 0,Y 181.915,Z 527.771,A -85,B 0,C 180,E1 -23102.381,E2 -23102.381} C_VEL
LIN {X 0,Y 178.332,Z 533.125,A -85,B 0,C 180,E1 -23105.557,E2 -23105.557} C_VEL
LIN {X 0,Y 175.297,Z 537.398,A -85,B 0,C 180,E1 -23108.85,E2 -23108.85} C_VEL
LIN {X 0,Y 173.469,Z 539.703,A -85,B 0,C 180,E1 -23111.089,E2 -23111.089} C_VEL
LIN {X 0,Y 171.946,Z 541.592,A -85,B 0,C 180,E1 -23113.376,E2 -23113.376} C_VEL
LIN {X 0,Y 170.05,Z 544.128,A -85,B 0,C 180,E1 -23118.075,E2 -23118.075} C_VEL
LIN {X 0,Y 169.09,Z 545.182,A -85,B 0,C 180,E1 -23122.838,E2 -23122.838} C_VEL
LIN {X 0,Y 168.954,Z 544.89,A -85,B 0,C 180,E1 -23126.693,E2 -23126.693} C_VEL
LIN {X 0,Y 169.197,Z 543.812,A -85,B 0,C 180,E1 -23130.001,E2 -23130.001} C_VEL
LIN {X 0,Y 169.024,Z 541.63,A -85,B 0,C 180,E1 -23133.693,E2 -23133.693} C_VEL
LIN {X 0,Y 169.222,Z 538.361,A -85,B 0,C 180,E1 -23137.401,E2 -23137.401} C_VEL
LIN {X 0,Y 169.727,Z 534.415,A -85,B 0,C 180,E1 -23140.74,E2 -23140.74} C_VEL
LIN {X 0,Y 170.911,Z 527.995,A -85,B 0,C 180,E1 -23144.893,E2 -23144.893} C_VEL
LIN {X 0,Y 171.679,Z 524.837,A -85,B 0,C 180,E1 -23146.569,E2 -23146.569} C_VEL
LIN {X 0,Y 171.854,Z 521.532,A -85,B 0,C 180,E1 -23148.201,E2 -23148.201} C_VEL
LIN {X 0,Y 170.503,Z 515.574,A -85,B 0,C 180,E1 -23150.82,E2 -23150.82} C_VEL
LIN {X 0,Y 169.362,Z 509,A -85,B 0,C 180,E1 -23153.307,E2 -23153.307} C_VEL
LIN {X 0,Y 169.86,Z 504.725,A -85,B 0,C 180,E1 -23154.682,E2 -23154.682} C_VEL
LIN {X 0,Y 171.727,Z 497.243,A -85,B 0,C 180,E1 -23156.756,E2 -23156.756} C_VEL
LIN {X 0,Y 171.695,Z 486.557,A -85,B 0,C 180,E1 -23159.42,E2 -23159.42} C_VEL
LIN {X 0,Y 171.133,Z 475.552,A -85,B 0,C 180,E1 -23161.743,E2 -23161.743} C_VEL
LIN {X 0,Y 169.973,Z 463.127,A -85,B 0,C 180,E1 -23163.948,E2 -23163.948} C_VEL
LIN {X 0,Y 167.983,Z 449.617,A -85,B 0,C 180,E1 -23165.918,E2 -23165.918} C_VEL
LIN {X 0,Y 165.854,Z 439.372,A -85,B 0,C 180,E1 -23167.241,E2 -23167.241} C_VEL
LIN {X 0,Y 165.781,Z 437.152,A -85,B 0,C 180,E1 -23170.263,E2 -23170.263} C_VEL
LIN {X 0,Y 165.32,Z 434.708,A -85,B 0,C 180,E1 -23173.722,E2 -23173.722} C_VEL
LIN {X 0,Y 164.715,Z 431.437,A -85,B 0,C 180,E1 -23178.597,E2 -23178.597} C_VEL
LIN {X 0,Y 164.472,Z 430.004,A -85,B 0,C 180,E1 -23181.008,E2 -23181.008} C_VEL
LIN {X 0,Y 164.334,Z 430.014,A -85,B 0,C 180,E1 -23186.222,E2 -23186.222} C_VEL
LIN {X 0,Y 164.408,Z 430.007,A -85,B 0,C 180,E1 -23189.138,E2 -23189.138} C_VEL
LIN {X 0,Y 164.419,Z 429.995,A -85,B 0,C 180,E1 -23194.694,E2 -23194.694} C_VEL
LIN {X 0,Y 164.487,Z 429.993,A -85,B 0,C 180,E1 -23200.051,E2 -23200.051} C_VEL
LIN {X 0,Y 164.556,Z 429.988,A -85,B 0,C 180,E1 -23205.152,E2 -23205.152} C_VEL
LIN {X 0,Y 164.811,Z 429.951,A -85,B 0,C 180,E1 -23210.179,E2 -23210.179} C_VEL
LIN {X 0,Y 164.854,Z 429.949,A -85,B 0,C 180,E1 -23212.652,E2 -23212.652} C_VEL
LIN {X 0,Y 165.051,Z 429.92,A -85,B 0,C 180,E1 -23217.559,E2 -23217.559} C_VEL
LIN {X 0,Y 165.296,Z 429.892,A -85,B 0,C 180,E1 -23220,E2 -23220} C_VEL
LIN {X 0,Y 164.773,Z 429.951,A -85,B 0,C 180,E1 -23224.893,E2 -23224.893} C_VEL
LIN {X 0,Y 164.853,Z 429.947,A -85,B 0,C 180,E1 -23227.348,E2 -23227.348} C_VEL
LIN {X 0,Y 164.756,Z 429.957,A -85,B 0,C 180,E1 -23231.152,E2 -23231.152} C_VEL
LIN {X 0,Y 164.486,Z 429.962,A -85,B 0,C 180,E1 -23237.403,E2 -23237.403} C_VEL
LIN {X 0,Y 164.476,Z 429.974,A -85,B 0,C 180,E1 -23239.989,E2 -23239.989} C_VEL
LIN {X 0,Y 164.396,Z 430.006,A -85,B 0,C 180,E1 -23246.134,E2 -23246.134} C_VEL
LIN {X 0,Y 164.378,Z 430,A -85,B 0,C 180,E1 -23251.228,E2 -23251.228} C_VEL
LIN {X 0,Y 164.296,Z 429.992,A -85,B 0,C 180,E1 -23256.789,E2 -23256.789} C_VEL
LIN {X 0,Y 164.292,Z 430.01,A -85,B 0,C 180,E1 -23259.916,E2 -23259.916} C_VEL
LIN {X 0,Y 164.281,Z 430.02,A -85,B 0,C 180,E1 -23263.341,E2 -23263.341} C_VEL
LIN {X 0,Y 164.294,Z 430.014,A -85,B 0,C 180,E1 -23266.808,E2 -23266.808} C_VEL
LIN {X 0,Y 164.307,Z 429.998,A -85,B 0,C 180,E1 -23270.347,E2 -23270.347} C_VEL
LIN {X 0,Y 164.345,Z 430.006,A -85,B 0,C 180,E1 -23274.342,E2 -23274.342} C_VEL
LIN {X 0,Y 164.393,Z 430.005,A -85,B 0,C 180,E1 -23279.134,E2 -23279.134} C_VEL
LIN {X 0,Y 164.418,Z 429.997,A -85,B 0,C 180,E1 -23284.694,E2 -23284.694} C_VEL
LIN {X 0,Y 164.486,Z 429.993,A -85,B 0,C 180,E1 -23290.05,E2 -23290.05} C_VEL
LIN {X 0,Y 164.555,Z 429.989,A -85,B 0,C 180,E1 -23295.151,E2 -23295.151} C_VEL
LIN {X 0,Y 164.855,Z 429.948,A -85,B 0,C 180,E1 -23300.181,E2 -23300.181} C_VEL
LIN {X 0,Y 164.864,Z 429.948,A -85,B 0,C 180,E1 -23302.652,E2 -23302.652} C_VEL
LIN {X 0,Y 165.051,Z 429.918,A -85,B 0,C 180,E1 -23307.559,E2 -23307.559} C_VEL
LIN {X 0,Y 165.293,Z 429.899,A -85,B 0,C 180,E1 -23309.999,E2 -23309.999} C_VEL
LIN {X 0,Y 164.605,Z 429.986,A -85,B 0,C 180,E1 -23315.819,E2 -23315.819} C_VEL
LIN {X 0,Y 167.668,Z 438.75,A -85,B 0,C 180,E1 -23317.223,E2 -23317.223} C_VEL
LIN {X 0,Y 170.566,Z 450.648,A -85,B 0,C 180,E1 -23319.187,E2 -23319.187} C_VEL
LIN {X 0,Y 172.696,Z 462.28,A -85,B 0,C 180,E1 -23321.412,E2 -23321.412} C_VEL
LIN {X 0,Y 174.164,Z 474.022,A -85,B 0,C 180,E1 -23324.01,E2 -23324.01} C_VEL
LIN {X 0,Y 174.45,Z 477.196,A -85,B 0,C 180,E1 -23324.788,E2 -23324.788} C_VEL
LIN {X 0,Y 171.656,Z 488.692,A -85,B 0,C 180,E1 -23327.574,E2 -23327.574} C_VEL
LIN {X 0,Y 168.994,Z 498.703,A -85,B 0,C 180,E1 -23330.7,E2 -23330.7} C_VEL
LIN {X 0,Y 166.514,Z 507.965,A -85,B 0,C 180,E1 -23334.386,E2 -23334.386} C_VEL
LIN {X 0,Y 164.655,Z 515.061,A -85,B 0,C 180,E1 -23338.002,E2 -23338.002} C_VEL
LIN {X 0,Y 163.208,Z 520.964,A -85,B 0,C 180,E1 -23341.836,E2 -23341.836} C_VEL
LIN {X 0,Y 162.219,Z 525.83,A -85,B 0,C 180,E1 -23345.964,E2 -23345.964} C_VEL
LIN {X 0,Y 161.745,Z 528.212,A -85,B 0,C 180,E1 -23348.545,E2 -23348.545} C_VEL
LIN {X 0,Y 161.435,Z 530.753,A -85,B 0,C 180,E1 -23352.261,E2 -23352.261} C_VEL
LIN {X 0,Y 161.598,Z 532.356,A -85,B 0,C 180,E1 -23355.905,E2 -23355.905} C_VEL
LIN {X 0,Y 162.627,Z 533.232,A -85,B 0,C 180,E1 -23361.065,E2 -23361.065} C_VEL
LIN {X 0,Y 163.882,Z 532.881,A -85,B 0,C 180,E1 -23364.566,E2 -23364.566} C_VEL
LIN {X 0,Y 166.563,Z 530.921,A -85,B 0,C 180,E1 -23369.58,E2 -23369.58} C_VEL
LIN {X 0,Y 168.874,Z 528.758,A -85,B 0,C 180,E1 -23372.756,E2 -23372.756} C_VEL
LIN {X 0,Y 172.944,Z 524.336,A -85,B 0,C 180,E1 -23377.12,E2 -23377.12} C_VEL
LIN {X 0,Y 176.536,Z 520.02,A -85,B 0,C 180,E1 -23380.164,E2 -23380.164} C_VEL
LIN {X 0,Y 181.617,Z 513.339,A -85,B 0,C 180,E1 -23383.708,E2 -23383.708} C_VEL
LIN {X 0,Y 187.108,Z 505.039,A -85,B 0,C 180,E1 -23386.976,E2 -23386.976} C_VEL
LIN {X 0,Y 190.811,Z 498.932,A -85,B 0,C 180,E1 -23388.885,E2 -23388.885} C_VEL
LIN {X 0,Y 191.629,Z 497.157,A -85,B 0,C 180,E1 -23389.434,E2 -23389.434} C_VEL
LIN {X 0,Y 192.54,Z 490.523,A -85,B 0,C 180,E1 -23392.133,E2 -23392.133} C_VEL
LIN {X 0,Y 192.617,Z 483.079,A -85,B 0,C 180,E1 -23395.291,E2 -23395.291} C_VEL
LIN {X 0,Y 192.116,Z 478.597,A -85,B 0,C 180,E1 -23397.379,E2 -23397.379} C_VEL
LIN {X 0,Y 190.331,Z 472.245,A -85,B 0,C 180,E1 -23401.009,E2 -23401.009} C_VEL
LIN {X 0,Y 189.264,Z 468.872,A -85,B 0,C 180,E1 -23403.148,E2 -23403.148} C_VEL
LIN {X 0,Y 186.912,Z 464.116,A -85,B 0,C 180,E1 -23407.344,E2 -23407.344} C_VEL
LIN {X 0,Y 184.602,Z 459.443,A -85,B 0,C 180,E1 -23413.205,E2 -23413.205} C_VEL
LIN {X 0,Y 183.159,Z 458.72,A -85,B 0,C 180,E1 -23417.877,E2 -23417.877} C_VEL
LIN {X 0,Y 182.877,Z 459.102,A -85,B 0,C 180,E1 -23422.735,E2 -23422.735} C_VEL
LIN {X 0,Y 183.691,Z 460.635,A -85,B 0,C 180,E1 -23427.33,E2 -23427.33} C_VEL
LIN {X 0,Y 184.398,Z 462.101,A -85,B 0,C 180,E1 -23429.701,E2 -23429.701} C_VEL
LIN {X 0,Y 186.681,Z 468.104,A -85,B 0,C 180,E1 -23435.381,E2 -23435.381} C_VEL
LIN {X 0,Y 188.599,Z 473.978,A -85,B 0,C 180,E1 -23439.308,E2 -23439.308} C_VEL
LIN {X 0,Y 189.481,Z 476.529,A -85,B 0,C 180,E1 -23440.843,E2 -23440.843} C_VEL
LIN {X 0,Y 191.035,Z 483.54,A -85,B 0,C 180,E1 -23444.347,E2 -23444.347} C_VEL
LIN {X 0,Y 191.335,Z 487.475,A -85,B 0,C 180,E1 -23445.956,E2 -23445.956} C_VEL
LIN {X 0,Y 190.756,Z 494.552,A -85,B 0,C 180,E1 -23448.459,E2 -23448.459} C_VEL
LIN {X 0,Y 189.281,Z 502.976,A -85,B 0,C 180,E1 -23451.39,E2 -23451.39} C_VEL
LIN {X 0,Y 187.258,Z 509.677,A -85,B 0,C 180,E1 -23453.765,E2 -23453.765} C_VEL
LIN {X 0,Y 186.128,Z 512.625,A -85,B 0,C 180,E1 -23454.844,E2 -23454.844} C_VEL
LIN {X 0,Y 181.012,Z 520.705,A -85,B 0,C 180,E1 -23457.735,E2 -23457.735} C_VEL
LIN {X 0,Y 175.687,Z 528.318,A -85,B 0,C 180,E1 -23461.313,E2 -23461.313} C_VEL
LIN {X 0,Y 171.898,Z 533.489,A -85,B 0,C 180,E1 -23464.579,E2 -23464.579} C_VEL
LIN {X 0,Y 168.679,Z 537.59,A -85,B 0,C 180,E1 -23467.978,E2 -23467.978} C_VEL
LIN {X 0,Y 166.758,Z 539.815,A -85,B 0,C 180,E1 -23470.297,E2 -23470.297} C_VEL
LIN {X 0,Y 165.138,Z 541.591,A -85,B 0,C 180,E1 -23472.669,E2 -23472.669} C_VEL
LIN {X 0,Y 163.091,Z 544,A -85,B 0,C 180,E1 -23477.558,E2 -23477.558} C_VEL
LIN {X 0,Y 162.019,Z 544.904,A -85,B 0,C 180,E1 -23482.524,E2 -23482.524} C_VEL
LIN {X 0,Y 161.926,Z 544.247,A -85,B 0,C 180,E1 -23487.513,E2 -23487.513} C_VEL
LIN {X 0,Y 162.117,Z 543.343,A -85,B 0,C 180,E1 -23490.001,E2 -23490.001} C_VEL
LIN {X 0,Y 161.939,Z 541.326,A -85,B 0,C 180,E1 -23493.452,E2 -23493.452} C_VEL
LIN {X 0,Y 162.147,Z 537.906,A -85,B 0,C 180,E1 -23497.472,E2 -23497.472} C_VEL
LIN {X 0,Y 162.728,Z 533.578,A -85,B 0,C 180,E1 -23501.208,E2 -23501.208} C_VEL
LIN {X 0,Y 163.769,Z 528.024,A -85,B 0,C 180,E1 -23504.922,E2 -23504.922} C_VEL
LIN {X 0,Y 165.559,Z 521.096,A -85,B 0,C 180,E1 -23508.566,E2 -23508.566} C_VEL
LIN {X 0,Y 167.754,Z 512.374,A -85,B 0,C 180,E1 -23512.152,E2 -23512.152} C_VEL
LIN {X 0,Y 169.86,Z 504.725,A -85,B 0,C 180,E1 -23514.682,E2 -23514.682} C_VEL
LIN {X 0,Y 170.241,Z 501.858,A -85,B 0,C 180,E1 -23515.555,E2 -23515.555} C_VEL
LIN {X 0,Y 169.627,Z 497.469,A -85,B 0,C 180,E1 -23516.886,E2 -23516.886} C_VEL
LIN {X 0,Y 168.176,Z 493.132,A -85,B 0,C 180,E1 -23518.2,E2 -23518.2} C_VEL
LIN {X 0,Y 165.055,Z 484.027,A -85,B 0,C 180,E1 -23520.768,E2 -23520.768} C_VEL
LIN {X 0,Y 164.622,Z 480.666,A -85,B 0,C 180,E1 -23521.556,E2 -23521.556} C_VEL
LIN {X 0,Y 163.831,Z 469.117,A -85,B 0,C 180,E1 -23523.896,E2 -23523.896} C_VEL
LIN {X 0,Y 162.502,Z 457.437,A -85,B 0,C 180,E1 -23525.873,E2 -23525.873} C_VEL
LIN {X 0,Y 160.335,Z 444.842,A -85,B 0,C 180,E1 -23527.665,E2 -23527.665} C_VEL
LIN {X 0,Y 158.807,Z 439.149,A -85,B 0,C 180,E1 -23528.487,E2 -23528.487} C_VEL
LIN {X 0,Y 158.334,Z 435.899,A -85,B 0,C 180,E1 -23533.205,E2 -23533.205} C_VEL
LIN {X 0,Y 157.542,Z 431.602,A -85,B 0,C 180,E1 -23539.879,E2 -23539.879} C_VEL
LIN {X 0,Y 157.428,Z 430.877,A -85,B 0,C 180,E1 -23541.318,E2 -23541.318} C_VEL
LIN {X 0,Y 157.304,Z 430.892,A -85,B 0,C 180,E1 -23548.091,E2 -23548.091} C_VEL
LIN {X 0,Y 157.324,Z 430.874,A -85,B 0,C 180,E1 -23553.466,E2 -23553.466} C_VEL
LIN {X 0,Y 157.397,Z 430.877,A -85,B 0,C 180,E1 -23559.667,E2 -23559.667} C_VEL
LIN {X 0,Y 157.481,Z 430.868,A -85,B 0,C 180,E1 -23564.468,E2 -23564.468} C_VEL
LIN {X 0,Y 157.737,Z 430.832,A -85,B 0,C 180,E1 -23569.734,E2 -23569.734} C_VEL
LIN {X 0,Y 157.811,Z 430.826,A -85,B 0,C 180,E1 -23572.322,E2 -23572.322} C_VEL
LIN {X 0,Y 158.258,Z 430.768,A -85,B 0,C 180,E1 -23580,E2 -23580} C_VEL
LIN {X 0,Y 157.811,Z 430.823,A -85,B 0,C 180,E1 -23587.678,E2 -23587.678} C_VEL
LIN {X 0,Y 157.685,Z 430.837,A -85,B 0,C 180,E1 -23591.32,E2 -23591.32} C_VEL
LIN {X 0,Y 157.464,Z 430.848,A -85,B 0,C 180,E1 -23595.533,E2 -23595.533} C_VEL
LIN {X 0,Y 157.372,Z 430.862,A -85,B 0,C 180,E1 -23600.932,E2 -23600.932} C_VEL
LIN {X 0,Y 157.317,Z 430.889,A -85,B 0,C 180,E1 -23606.685,E2 -23606.685} C_VEL
LIN {X 0,Y 157.277,Z 430.879,A -85,B 0,C 180,E1 -23612.427,E2 -23612.427} C_VEL
LIN {X 0,Y 157.269,Z 430.864,A -85,B 0,C 180,E1 -23616.449,E2 -23616.449} C_VEL
LIN {X 0,Y 157.194,Z 430.901,A -85,B 0,C 180,E1 -23622.116,E2 -23622.116} C_VEL
LIN {X 0,Y 157.214,Z 430.894,A -85,B 0,C 180,E1 -23627.89,E2 -23627.89} C_VEL
LIN {X 0,Y 157.285,Z 430.883,A -85,B 0,C 180,E1 -23633.543,E2 -23633.543} C_VEL
LIN {X 0,Y 157.297,Z 430.891,A -85,B 0,C 180,E1 -23638.094,E2 -23638.094} C_VEL
LIN {X 0,Y 157.324,Z 430.875,A -85,B 0,C 180,E1 -23643.466,E2 -23643.466} C_VEL
LIN {X 0,Y 157.396,Z 430.877,A -85,B 0,C 180,E1 -23649.667,E2 -23649.667} C_VEL
LIN {X 0,Y 157.48,Z 430.87,A -85,B 0,C 180,E1 -23654.468,E2 -23654.468} C_VEL
LIN {X 0,Y 157.774,Z 430.828,A -85,B 0,C 180,E1 -23659.735,E2 -23659.735} C_VEL
LIN {X 0,Y 157.826,Z 430.826,A -85,B 0,C 180,E1 -23662.322,E2 -23662.322} C_VEL
LIN {X 0,Y 158.252,Z 430.776,A -85,B 0,C 180,E1 -23669.999,E2 -23669.999} C_VEL
LIN {X 0,Y 157.647,Z 430.848,A -85,B 0,C 180,E1 -23674.634,E2 -23674.634} C_VEL
LIN {X 0,Y 158.664,Z 433.779,A -85,B 0,C 180,E1 -23675.121,E2 -23675.121} C_VEL
LIN {X 0,Y 161.137,Z 440.16,A -85,B 0,C 180,E1 -23676.259,E2 -23676.259} C_VEL
LIN {X 0,Y 164.099,Z 452.755,A -85,B 0,C 180,E1 -23678.496,E2 -23678.496} C_VEL
LIN {X 0,Y 166.139,Z 464.423,A -85,B 0,C 180,E1 -23680.872,E2 -23680.872} C_VEL
LIN {X 0,Y 167.276,Z 474.384,A -85,B 0,C 180,E1 -23683.205,E2 -23683.205} C_VEL
